// TwinCAT 3 PLC project TcoIoBeckhoffTests
// Title: TcoIoBeckhoffTests
// Company: Vortex.Library
// ProjectVersion: 1.19.1.1780
// ProgramVersion: 3.1.4024.12
// libraries:
//   Tc2_Standard, * (Beckhoff Automation GmbH)
//   Tc2_System, * (Beckhoff Automation GmbH)
//   Tc3_Module, * (Beckhoff Automation GmbH)
//   TcoCore, 1.19.1.1780 (Vortex.Library)
//   TcoIoBeckhoff, 1.19.1.1780 (Vortex.Library)
// project tree:
//   / PlcTask.TcTTO
//   POUs/ MAIN.TcPOU, tcc.TcPOU
//   DUTs/IO/PdoEntries/ Status_3D84275F.TcDUT (not stored), Ctrl_1EFB4D3B.TcDUT, Ctrl_71604E86.TcDUT, Status_B0753356.TcDUT, Status_F2CE6D91.TcDUT
//   DUTs/IO/PDOs/ COM_TxPDO_Map_Inputs_Channel_3801C95E.TcDUT, COM_RxPDO_Map_Outputs_Channel_EADA2E0D.TcDUT, WcState_9091E0EB.TcDUT, InfoData_32EB74EA.TcDUT (not stored), Channel_830843C1.TcDUT, InfoData_6F19DB2B.TcDUT, Channel_42CA91F7.TcDUT, AO_Outputs_Channel_BA7EBB7C.TcDUT, COM_Inputs_3801C95E.TcDUT, COM_Outputs_DEF408EC.TcDUT, PM_Inputs_Channel_2F868086.TcDUT, PM_Status_data_2A9514CB.TcDUT, PM_Outputs_Channel_E5FBDE30.TcDUT, AI_Standard_Channel_A8DF64E3.TcDUT, AI_Standard_4A394481.TcDUT, AI_Standard_Channel_4A394481.TcDUT
//   DUTs/IO/Boxes/ EL6002_81703A53.TcDUT, EL1809_32157CFD.TcDUT (not stored), EL2809_2B6483BD.TcDUT, EL4004_D2A7C9B7.TcDUT, EL6001_B592E1CA.TcDUT, EK1100_1FC0878B.TcDUT (not stored), EK1110_1FC0878B.TcDUT (not stored), EL3403_200C4240.TcDUT, EK1122_1FC0878B.TcDUT (not stored), EL3174_DCC78662.TcDUT (not stored), EL3011_353F32DF.TcDUT (not stored), EL2008_E2806B95.TcDUT, EL3024_C4269E32.TcDUT (not stored)
//   DUTs/IO/Devices/ SyncUnitTasks_1988CF1B.TcDUT, SyncUnits_13973095.TcDUT
//   DUTs/IO/Topology/ Term_1_EK1200_342ABB04.TcDUT (not stored), Device_1_EtherCAT_4442729B.TcDUT, Term_9_EK1100_B6B701E6.TcDUT, Term_17_EK1100_B932616E.TcDUT (not stored), Term_16_EK1122_E3300954.TcDUT (not stored), Term_14_EK1100_ED6DF06D.TcDUT (not stored), Device_4_EtherCAT_7DA382B8.TcDUT
//   GVLs/ GVL_iXlinker.TcGVL
// (motion and I/O tree: see PLC project tcoiobeckhoff)
// real-time tasks:
//   TASK PlcTask: cycle T#10ms, priority 20, ADS port 350
//   TASK PlcTask1: cycle T#10ms, priority 21, ADS port 351
//   TASK PlcTask2: cycle T#10ms, priority 22, ADS port 352
// variable links:
//   TcoIoBeckhoffTests/TcoIoBeckhoffTests Instance <-> Device 1 (EtherCAT)
//     PlcTask Inputs/GVL_iXlinker.Device_1_EtherCAT.InfoData.AmsNetId <-> InfoData/AmsNetId
//     PlcTask Inputs/GVL_iXlinker.Device_1_EtherCAT.InfoData.CfgSlaveCount <-> InfoData/CfgSlaveCount
//     PlcTask Inputs/GVL_iXlinker.Device_1_EtherCAT.InfoData.ChangeCount <-> InfoData/ChangeCount
//     PlcTask Inputs/GVL_iXlinker.Device_1_EtherCAT.InfoData.DevId <-> InfoData/DevId
//     PlcTask Inputs/GVL_iXlinker.Device_1_EtherCAT.Inputs.DevState <-> Inputs/DevState
//     PlcTask Inputs/GVL_iXlinker.Device_1_EtherCAT.Inputs.Frm0InputToggle <-> Inputs/Frm0InputToggle
//     PlcTask Inputs/GVL_iXlinker.Device_1_EtherCAT.Inputs.Frm0State <-> Inputs/Frm0State
//     PlcTask Inputs/GVL_iXlinker.Device_1_EtherCAT.Inputs.Frm0WcState <-> Inputs/Frm0WcState
//     PlcTask Inputs/GVL_iXlinker.Device_1_EtherCAT.Inputs.SlaveCount <-> Inputs/SlaveCount
//     PlcTask Inputs/GVL_iXlinker.Device_1_EtherCAT.SyncUnits._default.PlcTask1.InfoData.ObjectId <-> SyncUnits/<default>/PlcTask1/InfoData/ObjectId
//     PlcTask Inputs/GVL_iXlinker.Device_1_EtherCAT.SyncUnits._default.PlcTask1.InfoData.SlaveCount <-> SyncUnits/<default>/PlcTask1/InfoData/SlaveCount
//     PlcTask Inputs/GVL_iXlinker.Device_1_EtherCAT.SyncUnits._default.PlcTask1.InfoData.State <-> SyncUnits/<default>/PlcTask1/InfoData/State
//     PlcTask Inputs/GVL_iXlinker.Device_1_EtherCAT.SyncUnits._default.PlcTask1.WcState.WcState <-> SyncUnits/<default>/PlcTask1/WcState/WcState
//     PlcTask Outputs/GVL_iXlinker.Device_1_EtherCAT.Outputs.DevCtrl <-> Outputs/DevCtrl
//     PlcTask Outputs/GVL_iXlinker.Device_1_EtherCAT.Outputs.Frm0Ctrl <-> Outputs/Frm0Ctrl
//     PlcTask Outputs/GVL_iXlinker.Device_1_EtherCAT.Outputs.Frm0WcCtrl <-> Outputs/Frm0WcCtrl
//   TcoIoBeckhoffTests/TcoIoBeckhoffTests Instance <-> Device 1 (EtherCAT)/Term 1 (EK1200)/Term 2 (EL6002)
//     PlcTask Inputs/GVL_iXlinker.Device_1_EtherCAT.Term_1_EK1200.Term_2_EL6002.COM_TxPDO_Map_Inputs_Channel_1.Data_In[0] <-> COM TxPDO-Map Inputs Channel 1/Data In 0
//     PlcTask Inputs/GVL_iXlinker.Device_1_EtherCAT.Term_1_EK1200.Term_2_EL6002.COM_TxPDO_Map_Inputs_Channel_1.Data_In[10] <-> COM TxPDO-Map Inputs Channel 1/Data In 10
//     PlcTask Inputs/GVL_iXlinker.Device_1_EtherCAT.Term_1_EK1200.Term_2_EL6002.COM_TxPDO_Map_Inputs_Channel_1.Data_In[11] <-> COM TxPDO-Map Inputs Channel 1/Data In 11
//     PlcTask Inputs/GVL_iXlinker.Device_1_EtherCAT.Term_1_EK1200.Term_2_EL6002.COM_TxPDO_Map_Inputs_Channel_1.Data_In[12] <-> COM TxPDO-Map Inputs Channel 1/Data In 12
//     PlcTask Inputs/GVL_iXlinker.Device_1_EtherCAT.Term_1_EK1200.Term_2_EL6002.COM_TxPDO_Map_Inputs_Channel_1.Data_In[13] <-> COM TxPDO-Map Inputs Channel 1/Data In 13
//     PlcTask Inputs/GVL_iXlinker.Device_1_EtherCAT.Term_1_EK1200.Term_2_EL6002.COM_TxPDO_Map_Inputs_Channel_1.Data_In[14] <-> COM TxPDO-Map Inputs Channel 1/Data In 14
//     PlcTask Inputs/GVL_iXlinker.Device_1_EtherCAT.Term_1_EK1200.Term_2_EL6002.COM_TxPDO_Map_Inputs_Channel_1.Data_In[15] <-> COM TxPDO-Map Inputs Channel 1/Data In 15
//     PlcTask Inputs/GVL_iXlinker.Device_1_EtherCAT.Term_1_EK1200.Term_2_EL6002.COM_TxPDO_Map_Inputs_Channel_1.Data_In[16] <-> COM TxPDO-Map Inputs Channel 1/Data In 16
//     PlcTask Inputs/GVL_iXlinker.Device_1_EtherCAT.Term_1_EK1200.Term_2_EL6002.COM_TxPDO_Map_Inputs_Channel_1.Data_In[17] <-> COM TxPDO-Map Inputs Channel 1/Data In 17
//     PlcTask Inputs/GVL_iXlinker.Device_1_EtherCAT.Term_1_EK1200.Term_2_EL6002.COM_TxPDO_Map_Inputs_Channel_1.Data_In[18] <-> COM TxPDO-Map Inputs Channel 1/Data In 18
//     PlcTask Inputs/GVL_iXlinker.Device_1_EtherCAT.Term_1_EK1200.Term_2_EL6002.COM_TxPDO_Map_Inputs_Channel_1.Data_In[19] <-> COM TxPDO-Map Inputs Channel 1/Data In 19
//     PlcTask Inputs/GVL_iXlinker.Device_1_EtherCAT.Term_1_EK1200.Term_2_EL6002.COM_TxPDO_Map_Inputs_Channel_1.Data_In[1] <-> COM TxPDO-Map Inputs Channel 1/Data In 1
//     PlcTask Inputs/GVL_iXlinker.Device_1_EtherCAT.Term_1_EK1200.Term_2_EL6002.COM_TxPDO_Map_Inputs_Channel_1.Data_In[20] <-> COM TxPDO-Map Inputs Channel 1/Data In 20
//     PlcTask Inputs/GVL_iXlinker.Device_1_EtherCAT.Term_1_EK1200.Term_2_EL6002.COM_TxPDO_Map_Inputs_Channel_1.Data_In[21] <-> COM TxPDO-Map Inputs Channel 1/Data In 21
//     PlcTask Inputs/GVL_iXlinker.Device_1_EtherCAT.Term_1_EK1200.Term_2_EL6002.COM_TxPDO_Map_Inputs_Channel_1.Data_In[2] <-> COM TxPDO-Map Inputs Channel 1/Data In 2
//     PlcTask Inputs/GVL_iXlinker.Device_1_EtherCAT.Term_1_EK1200.Term_2_EL6002.COM_TxPDO_Map_Inputs_Channel_1.Data_In[3] <-> COM TxPDO-Map Inputs Channel 1/Data In 3
//     PlcTask Inputs/GVL_iXlinker.Device_1_EtherCAT.Term_1_EK1200.Term_2_EL6002.COM_TxPDO_Map_Inputs_Channel_1.Data_In[4] <-> COM TxPDO-Map Inputs Channel 1/Data In 4
//     PlcTask Inputs/GVL_iXlinker.Device_1_EtherCAT.Term_1_EK1200.Term_2_EL6002.COM_TxPDO_Map_Inputs_Channel_1.Data_In[5] <-> COM TxPDO-Map Inputs Channel 1/Data In 5
//     PlcTask Inputs/GVL_iXlinker.Device_1_EtherCAT.Term_1_EK1200.Term_2_EL6002.COM_TxPDO_Map_Inputs_Channel_1.Data_In[6] <-> COM TxPDO-Map Inputs Channel 1/Data In 6
//     PlcTask Inputs/GVL_iXlinker.Device_1_EtherCAT.Term_1_EK1200.Term_2_EL6002.COM_TxPDO_Map_Inputs_Channel_1.Data_In[7] <-> COM TxPDO-Map Inputs Channel 1/Data In 7
//     PlcTask Inputs/GVL_iXlinker.Device_1_EtherCAT.Term_1_EK1200.Term_2_EL6002.COM_TxPDO_Map_Inputs_Channel_1.Data_In[8] <-> COM TxPDO-Map Inputs Channel 1/Data In 8
//     PlcTask Inputs/GVL_iXlinker.Device_1_EtherCAT.Term_1_EK1200.Term_2_EL6002.COM_TxPDO_Map_Inputs_Channel_1.Data_In[9] <-> COM TxPDO-Map Inputs Channel 1/Data In 9
//     PlcTask Inputs/GVL_iXlinker.Device_1_EtherCAT.Term_1_EK1200.Term_2_EL6002.COM_TxPDO_Map_Inputs_Channel_2.Data_In[0] <-> COM TxPDO-Map Inputs Channel 2/Data In 0
//     PlcTask Inputs/GVL_iXlinker.Device_1_EtherCAT.Term_1_EK1200.Term_2_EL6002.COM_TxPDO_Map_Inputs_Channel_2.Data_In[10] <-> COM TxPDO-Map Inputs Channel 2/Data In 10
//     PlcTask Inputs/GVL_iXlinker.Device_1_EtherCAT.Term_1_EK1200.Term_2_EL6002.COM_TxPDO_Map_Inputs_Channel_2.Data_In[11] <-> COM TxPDO-Map Inputs Channel 2/Data In 11
//     PlcTask Inputs/GVL_iXlinker.Device_1_EtherCAT.Term_1_EK1200.Term_2_EL6002.COM_TxPDO_Map_Inputs_Channel_2.Data_In[12] <-> COM TxPDO-Map Inputs Channel 2/Data In 12
//     PlcTask Inputs/GVL_iXlinker.Device_1_EtherCAT.Term_1_EK1200.Term_2_EL6002.COM_TxPDO_Map_Inputs_Channel_2.Data_In[13] <-> COM TxPDO-Map Inputs Channel 2/Data In 13
//     PlcTask Inputs/GVL_iXlinker.Device_1_EtherCAT.Term_1_EK1200.Term_2_EL6002.COM_TxPDO_Map_Inputs_Channel_2.Data_In[14] <-> COM TxPDO-Map Inputs Channel 2/Data In 14
//     PlcTask Inputs/GVL_iXlinker.Device_1_EtherCAT.Term_1_EK1200.Term_2_EL6002.COM_TxPDO_Map_Inputs_Channel_2.Data_In[15] <-> COM TxPDO-Map Inputs Channel 2/Data In 15
//     PlcTask Inputs/GVL_iXlinker.Device_1_EtherCAT.Term_1_EK1200.Term_2_EL6002.COM_TxPDO_Map_Inputs_Channel_2.Data_In[16] <-> COM TxPDO-Map Inputs Channel 2/Data In 16
//     PlcTask Inputs/GVL_iXlinker.Device_1_EtherCAT.Term_1_EK1200.Term_2_EL6002.COM_TxPDO_Map_Inputs_Channel_2.Data_In[17] <-> COM TxPDO-Map Inputs Channel 2/Data In 17
//     PlcTask Inputs/GVL_iXlinker.Device_1_EtherCAT.Term_1_EK1200.Term_2_EL6002.COM_TxPDO_Map_Inputs_Channel_2.Data_In[18] <-> COM TxPDO-Map Inputs Channel 2/Data In 18
//     PlcTask Inputs/GVL_iXlinker.Device_1_EtherCAT.Term_1_EK1200.Term_2_EL6002.COM_TxPDO_Map_Inputs_Channel_2.Data_In[19] <-> COM TxPDO-Map Inputs Channel 2/Data In 19
//     PlcTask Inputs/GVL_iXlinker.Device_1_EtherCAT.Term_1_EK1200.Term_2_EL6002.COM_TxPDO_Map_Inputs_Channel_2.Data_In[1] <-> COM TxPDO-Map Inputs Channel 2/Data In 1
//     PlcTask Inputs/GVL_iXlinker.Device_1_EtherCAT.Term_1_EK1200.Term_2_EL6002.COM_TxPDO_Map_Inputs_Channel_2.Data_In[20] <-> COM TxPDO-Map Inputs Channel 2/Data In 20
//     PlcTask Inputs/GVL_iXlinker.Device_1_EtherCAT.Term_1_EK1200.Term_2_EL6002.COM_TxPDO_Map_Inputs_Channel_2.Data_In[21] <-> COM TxPDO-Map Inputs Channel 2/Data In 21
//     PlcTask Inputs/GVL_iXlinker.Device_1_EtherCAT.Term_1_EK1200.Term_2_EL6002.COM_TxPDO_Map_Inputs_Channel_2.Data_In[2] <-> COM TxPDO-Map Inputs Channel 2/Data In 2
//     PlcTask Inputs/GVL_iXlinker.Device_1_EtherCAT.Term_1_EK1200.Term_2_EL6002.COM_TxPDO_Map_Inputs_Channel_2.Data_In[3] <-> COM TxPDO-Map Inputs Channel 2/Data In 3
//     PlcTask Inputs/GVL_iXlinker.Device_1_EtherCAT.Term_1_EK1200.Term_2_EL6002.COM_TxPDO_Map_Inputs_Channel_2.Data_In[4] <-> COM TxPDO-Map Inputs Channel 2/Data In 4
//     PlcTask Inputs/GVL_iXlinker.Device_1_EtherCAT.Term_1_EK1200.Term_2_EL6002.COM_TxPDO_Map_Inputs_Channel_2.Data_In[5] <-> COM TxPDO-Map Inputs Channel 2/Data In 5
//     PlcTask Inputs/GVL_iXlinker.Device_1_EtherCAT.Term_1_EK1200.Term_2_EL6002.COM_TxPDO_Map_Inputs_Channel_2.Data_In[6] <-> COM TxPDO-Map Inputs Channel 2/Data In 6
//     PlcTask Inputs/GVL_iXlinker.Device_1_EtherCAT.Term_1_EK1200.Term_2_EL6002.COM_TxPDO_Map_Inputs_Channel_2.Data_In[7] <-> COM TxPDO-Map Inputs Channel 2/Data In 7
//     PlcTask Inputs/GVL_iXlinker.Device_1_EtherCAT.Term_1_EK1200.Term_2_EL6002.COM_TxPDO_Map_Inputs_Channel_2.Data_In[8] <-> COM TxPDO-Map Inputs Channel 2/Data In 8
//     PlcTask Inputs/GVL_iXlinker.Device_1_EtherCAT.Term_1_EK1200.Term_2_EL6002.COM_TxPDO_Map_Inputs_Channel_2.Data_In[9] <-> COM TxPDO-Map Inputs Channel 2/Data In 9
//     PlcTask Inputs/GVL_iXlinker.Device_1_EtherCAT.Term_1_EK1200.Term_2_EL6002.COM_TxPDO_Map_Inputs_Channel_1.Status/Buffer_full <-> COM TxPDO-Map Inputs Channel 1/Status/Buffer full
//     PlcTask Inputs/GVL_iXlinker.Device_1_EtherCAT.Term_1_EK1200.Term_2_EL6002.COM_TxPDO_Map_Inputs_Channel_2.Status/Buffer_full <-> COM TxPDO-Map Inputs Channel 2/Status/Buffer full
//     PlcTask Inputs/GVL_iXlinker.Device_1_EtherCAT.Term_1_EK1200.Term_2_EL6002.COM_TxPDO_Map_Inputs_Channel_1.Status/Framing_error <-> COM TxPDO-Map Inputs Channel 1/Status/Framing error
//     PlcTask Inputs/GVL_iXlinker.Device_1_EtherCAT.Term_1_EK1200.Term_2_EL6002.COM_TxPDO_Map_Inputs_Channel_2.Status/Framing_error <-> COM TxPDO-Map Inputs Channel 2/Status/Framing error
//     PlcTask Inputs/GVL_iXlinker.Device_1_EtherCAT.Term_1_EK1200.Term_2_EL6002.COM_TxPDO_Map_Inputs_Channel_1.Status/Init_accepted <-> COM TxPDO-Map Inputs Channel 1/Status/Init accepted
//     PlcTask Inputs/GVL_iXlinker.Device_1_EtherCAT.Term_1_EK1200.Term_2_EL6002.COM_TxPDO_Map_Inputs_Channel_2.Status/Init_accepted <-> COM TxPDO-Map Inputs Channel 2/Status/Init accepted
//     PlcTask Inputs/GVL_iXlinker.Device_1_EtherCAT.Term_1_EK1200.Term_2_EL6002.COM_TxPDO_Map_Inputs_Channel_1.Status/Input_length <-> COM TxPDO-Map Inputs Channel 1/Status/Input length
//     PlcTask Inputs/GVL_iXlinker.Device_1_EtherCAT.Term_1_EK1200.Term_2_EL6002.COM_TxPDO_Map_Inputs_Channel_2.Status/Input_length <-> COM TxPDO-Map Inputs Channel 2/Status/Input length
//     PlcTask Inputs/GVL_iXlinker.Device_1_EtherCAT.Term_1_EK1200.Term_2_EL6002.COM_TxPDO_Map_Inputs_Channel_1.Status/Overrun_error <-> COM TxPDO-Map Inputs Channel 1/Status/Overrun error
//     PlcTask Inputs/GVL_iXlinker.Device_1_EtherCAT.Term_1_EK1200.Term_2_EL6002.COM_TxPDO_Map_Inputs_Channel_2.Status/Overrun_error <-> COM TxPDO-Map Inputs Channel 2/Status/Overrun error
//     PlcTask Inputs/GVL_iXlinker.Device_1_EtherCAT.Term_1_EK1200.Term_2_EL6002.COM_TxPDO_Map_Inputs_Channel_1.Status/Parity_error <-> COM TxPDO-Map Inputs Channel 1/Status/Parity error
//     PlcTask Inputs/GVL_iXlinker.Device_1_EtherCAT.Term_1_EK1200.Term_2_EL6002.COM_TxPDO_Map_Inputs_Channel_2.Status/Parity_error <-> COM TxPDO-Map Inputs Channel 2/Status/Parity error
//     PlcTask Inputs/GVL_iXlinker.Device_1_EtherCAT.Term_1_EK1200.Term_2_EL6002.COM_TxPDO_Map_Inputs_Channel_1.Status/Receive_request <-> COM TxPDO-Map Inputs Channel 1/Status/Receive request
//     PlcTask Inputs/GVL_iXlinker.Device_1_EtherCAT.Term_1_EK1200.Term_2_EL6002.COM_TxPDO_Map_Inputs_Channel_2.Status/Receive_request <-> COM TxPDO-Map Inputs Channel 2/Status/Receive request
//     PlcTask Inputs/GVL_iXlinker.Device_1_EtherCAT.Term_1_EK1200.Term_2_EL6002.COM_TxPDO_Map_Inputs_Channel_1.Status/Transmit_accepted <-> COM TxPDO-Map Inputs Channel 1/Status/Transmit accepted
//     PlcTask Inputs/GVL_iXlinker.Device_1_EtherCAT.Term_1_EK1200.Term_2_EL6002.COM_TxPDO_Map_Inputs_Channel_2.Status/Transmit_accepted <-> COM TxPDO-Map Inputs Channel 2/Status/Transmit accepted
//     PlcTask Inputs/GVL_iXlinker.Device_1_EtherCAT.Term_1_EK1200.Term_2_EL6002.InfoData.State <-> InfoData/State
//     PlcTask Inputs/GVL_iXlinker.Device_1_EtherCAT.Term_1_EK1200.Term_2_EL6002.WcState.InputToggle <-> WcState/InputToggle
//     PlcTask Inputs/GVL_iXlinker.Device_1_EtherCAT.Term_1_EK1200.Term_2_EL6002.WcState.WcState <-> WcState/WcState
//     PlcTask Outputs/GVL_iXlinker.Device_1_EtherCAT.Term_1_EK1200.Term_2_EL6002.COM_RxPDO_Map_Outputs_Channel_1.Ctrl/Init_request <-> COM RxPDO-Map Outputs Channel 1/Ctrl/Init request
//     PlcTask Outputs/GVL_iXlinker.Device_1_EtherCAT.Term_1_EK1200.Term_2_EL6002.COM_RxPDO_Map_Outputs_Channel_2.Ctrl/Init_request <-> COM RxPDO-Map Outputs Channel 2/Ctrl/Init request
//     PlcTask Outputs/GVL_iXlinker.Device_1_EtherCAT.Term_1_EK1200.Term_2_EL6002.COM_RxPDO_Map_Outputs_Channel_1.Ctrl/Output_length <-> COM RxPDO-Map Outputs Channel 1/Ctrl/Output length
//     PlcTask Outputs/GVL_iXlinker.Device_1_EtherCAT.Term_1_EK1200.Term_2_EL6002.COM_RxPDO_Map_Outputs_Channel_2.Ctrl/Output_length <-> COM RxPDO-Map Outputs Channel 2/Ctrl/Output length
//     PlcTask Outputs/GVL_iXlinker.Device_1_EtherCAT.Term_1_EK1200.Term_2_EL6002.COM_RxPDO_Map_Outputs_Channel_1.Ctrl/Receive_accepted <-> COM RxPDO-Map Outputs Channel 1/Ctrl/Receive accepted
//     PlcTask Outputs/GVL_iXlinker.Device_1_EtherCAT.Term_1_EK1200.Term_2_EL6002.COM_RxPDO_Map_Outputs_Channel_2.Ctrl/Receive_accepted <-> COM RxPDO-Map Outputs Channel 2/Ctrl/Receive accepted
//     PlcTask Outputs/GVL_iXlinker.Device_1_EtherCAT.Term_1_EK1200.Term_2_EL6002.COM_RxPDO_Map_Outputs_Channel_1.Ctrl/Send_continuous <-> COM RxPDO-Map Outputs Channel 1/Ctrl/Send continuous
//     PlcTask Outputs/GVL_iXlinker.Device_1_EtherCAT.Term_1_EK1200.Term_2_EL6002.COM_RxPDO_Map_Outputs_Channel_2.Ctrl/Send_continuous <-> COM RxPDO-Map Outputs Channel 2/Ctrl/Send continuous
//     PlcTask Outputs/GVL_iXlinker.Device_1_EtherCAT.Term_1_EK1200.Term_2_EL6002.COM_RxPDO_Map_Outputs_Channel_1.Ctrl/Transmit_request <-> COM RxPDO-Map Outputs Channel 1/Ctrl/Transmit request
//     PlcTask Outputs/GVL_iXlinker.Device_1_EtherCAT.Term_1_EK1200.Term_2_EL6002.COM_RxPDO_Map_Outputs_Channel_2.Ctrl/Transmit_request <-> COM RxPDO-Map Outputs Channel 2/Ctrl/Transmit request
//     PlcTask Outputs/GVL_iXlinker.Device_1_EtherCAT.Term_1_EK1200.Term_2_EL6002.COM_RxPDO_Map_Outputs_Channel_1.Data_Out[0] <-> COM RxPDO-Map Outputs Channel 1/Data Out 0
//     PlcTask Outputs/GVL_iXlinker.Device_1_EtherCAT.Term_1_EK1200.Term_2_EL6002.COM_RxPDO_Map_Outputs_Channel_1.Data_Out[10] <-> COM RxPDO-Map Outputs Channel 1/Data Out 10
//     PlcTask Outputs/GVL_iXlinker.Device_1_EtherCAT.Term_1_EK1200.Term_2_EL6002.COM_RxPDO_Map_Outputs_Channel_1.Data_Out[11] <-> COM RxPDO-Map Outputs Channel 1/Data Out 11
//     PlcTask Outputs/GVL_iXlinker.Device_1_EtherCAT.Term_1_EK1200.Term_2_EL6002.COM_RxPDO_Map_Outputs_Channel_1.Data_Out[12] <-> COM RxPDO-Map Outputs Channel 1/Data Out 12
//     PlcTask Outputs/GVL_iXlinker.Device_1_EtherCAT.Term_1_EK1200.Term_2_EL6002.COM_RxPDO_Map_Outputs_Channel_1.Data_Out[13] <-> COM RxPDO-Map Outputs Channel 1/Data Out 13
//     PlcTask Outputs/GVL_iXlinker.Device_1_EtherCAT.Term_1_EK1200.Term_2_EL6002.COM_RxPDO_Map_Outputs_Channel_1.Data_Out[14] <-> COM RxPDO-Map Outputs Channel 1/Data Out 14
//     PlcTask Outputs/GVL_iXlinker.Device_1_EtherCAT.Term_1_EK1200.Term_2_EL6002.COM_RxPDO_Map_Outputs_Channel_1.Data_Out[15] <-> COM RxPDO-Map Outputs Channel 1/Data Out 15
//     PlcTask Outputs/GVL_iXlinker.Device_1_EtherCAT.Term_1_EK1200.Term_2_EL6002.COM_RxPDO_Map_Outputs_Channel_1.Data_Out[16] <-> COM RxPDO-Map Outputs Channel 1/Data Out 16
//     PlcTask Outputs/GVL_iXlinker.Device_1_EtherCAT.Term_1_EK1200.Term_2_EL6002.COM_RxPDO_Map_Outputs_Channel_1.Data_Out[17] <-> COM RxPDO-Map Outputs Channel 1/Data Out 17
//     PlcTask Outputs/GVL_iXlinker.Device_1_EtherCAT.Term_1_EK1200.Term_2_EL6002.COM_RxPDO_Map_Outputs_Channel_1.Data_Out[18] <-> COM RxPDO-Map Outputs Channel 1/Data Out 18
//     PlcTask Outputs/GVL_iXlinker.Device_1_EtherCAT.Term_1_EK1200.Term_2_EL6002.COM_RxPDO_Map_Outputs_Channel_1.Data_Out[19] <-> COM RxPDO-Map Outputs Channel 1/Data Out 19
//     PlcTask Outputs/GVL_iXlinker.Device_1_EtherCAT.Term_1_EK1200.Term_2_EL6002.COM_RxPDO_Map_Outputs_Channel_1.Data_Out[1] <-> COM RxPDO-Map Outputs Channel 1/Data Out 1
//     PlcTask Outputs/GVL_iXlinker.Device_1_EtherCAT.Term_1_EK1200.Term_2_EL6002.COM_RxPDO_Map_Outputs_Channel_1.Data_Out[20] <-> COM RxPDO-Map Outputs Channel 1/Data Out 20
//     PlcTask Outputs/GVL_iXlinker.Device_1_EtherCAT.Term_1_EK1200.Term_2_EL6002.COM_RxPDO_Map_Outputs_Channel_1.Data_Out[21] <-> COM RxPDO-Map Outputs Channel 1/Data Out 21
//     PlcTask Outputs/GVL_iXlinker.Device_1_EtherCAT.Term_1_EK1200.Term_2_EL6002.COM_RxPDO_Map_Outputs_Channel_1.Data_Out[2] <-> COM RxPDO-Map Outputs Channel 1/Data Out 2
//     PlcTask Outputs/GVL_iXlinker.Device_1_EtherCAT.Term_1_EK1200.Term_2_EL6002.COM_RxPDO_Map_Outputs_Channel_1.Data_Out[3] <-> COM RxPDO-Map Outputs Channel 1/Data Out 3
//     PlcTask Outputs/GVL_iXlinker.Device_1_EtherCAT.Term_1_EK1200.Term_2_EL6002.COM_RxPDO_Map_Outputs_Channel_1.Data_Out[4] <-> COM RxPDO-Map Outputs Channel 1/Data Out 4
//     PlcTask Outputs/GVL_iXlinker.Device_1_EtherCAT.Term_1_EK1200.Term_2_EL6002.COM_RxPDO_Map_Outputs_Channel_1.Data_Out[5] <-> COM RxPDO-Map Outputs Channel 1/Data Out 5
//     PlcTask Outputs/GVL_iXlinker.Device_1_EtherCAT.Term_1_EK1200.Term_2_EL6002.COM_RxPDO_Map_Outputs_Channel_1.Data_Out[6] <-> COM RxPDO-Map Outputs Channel 1/Data Out 6
//     PlcTask Outputs/GVL_iXlinker.Device_1_EtherCAT.Term_1_EK1200.Term_2_EL6002.COM_RxPDO_Map_Outputs_Channel_1.Data_Out[7] <-> COM RxPDO-Map Outputs Channel 1/Data Out 7
//     PlcTask Outputs/GVL_iXlinker.Device_1_EtherCAT.Term_1_EK1200.Term_2_EL6002.COM_RxPDO_Map_Outputs_Channel_1.Data_Out[8] <-> COM RxPDO-Map Outputs Channel 1/Data Out 8
//     PlcTask Outputs/GVL_iXlinker.Device_1_EtherCAT.Term_1_EK1200.Term_2_EL6002.COM_RxPDO_Map_Outputs_Channel_1.Data_Out[9] <-> COM RxPDO-Map Outputs Channel 1/Data Out 9
//     PlcTask Outputs/GVL_iXlinker.Device_1_EtherCAT.Term_1_EK1200.Term_2_EL6002.COM_RxPDO_Map_Outputs_Channel_2.Data_Out[0] <-> COM RxPDO-Map Outputs Channel 2/Data Out 0
//     PlcTask Outputs/GVL_iXlinker.Device_1_EtherCAT.Term_1_EK1200.Term_2_EL6002.COM_RxPDO_Map_Outputs_Channel_2.Data_Out[10] <-> COM RxPDO-Map Outputs Channel 2/Data Out 10
//     PlcTask Outputs/GVL_iXlinker.Device_1_EtherCAT.Term_1_EK1200.Term_2_EL6002.COM_RxPDO_Map_Outputs_Channel_2.Data_Out[11] <-> COM RxPDO-Map Outputs Channel 2/Data Out 11
//     PlcTask Outputs/GVL_iXlinker.Device_1_EtherCAT.Term_1_EK1200.Term_2_EL6002.COM_RxPDO_Map_Outputs_Channel_2.Data_Out[12] <-> COM RxPDO-Map Outputs Channel 2/Data Out 12
//     PlcTask Outputs/GVL_iXlinker.Device_1_EtherCAT.Term_1_EK1200.Term_2_EL6002.COM_RxPDO_Map_Outputs_Channel_2.Data_Out[13] <-> COM RxPDO-Map Outputs Channel 2/Data Out 13
//     PlcTask Outputs/GVL_iXlinker.Device_1_EtherCAT.Term_1_EK1200.Term_2_EL6002.COM_RxPDO_Map_Outputs_Channel_2.Data_Out[14] <-> COM RxPDO-Map Outputs Channel 2/Data Out 14
//     PlcTask Outputs/GVL_iXlinker.Device_1_EtherCAT.Term_1_EK1200.Term_2_EL6002.COM_RxPDO_Map_Outputs_Channel_2.Data_Out[15] <-> COM RxPDO-Map Outputs Channel 2/Data Out 15
//     PlcTask Outputs/GVL_iXlinker.Device_1_EtherCAT.Term_1_EK1200.Term_2_EL6002.COM_RxPDO_Map_Outputs_Channel_2.Data_Out[16] <-> COM RxPDO-Map Outputs Channel 2/Data Out 16
//     PlcTask Outputs/GVL_iXlinker.Device_1_EtherCAT.Term_1_EK1200.Term_2_EL6002.COM_RxPDO_Map_Outputs_Channel_2.Data_Out[17] <-> COM RxPDO-Map Outputs Channel 2/Data Out 17
//     PlcTask Outputs/GVL_iXlinker.Device_1_EtherCAT.Term_1_EK1200.Term_2_EL6002.COM_RxPDO_Map_Outputs_Channel_2.Data_Out[18] <-> COM RxPDO-Map Outputs Channel 2/Data Out 18
//     PlcTask Outputs/GVL_iXlinker.Device_1_EtherCAT.Term_1_EK1200.Term_2_EL6002.COM_RxPDO_Map_Outputs_Channel_2.Data_Out[19] <-> COM RxPDO-Map Outputs Channel 2/Data Out 19
//     PlcTask Outputs/GVL_iXlinker.Device_1_EtherCAT.Term_1_EK1200.Term_2_EL6002.COM_RxPDO_Map_Outputs_Channel_2.Data_Out[1] <-> COM RxPDO-Map Outputs Channel 2/Data Out 1
//     PlcTask Outputs/GVL_iXlinker.Device_1_EtherCAT.Term_1_EK1200.Term_2_EL6002.COM_RxPDO_Map_Outputs_Channel_2.Data_Out[20] <-> COM RxPDO-Map Outputs Channel 2/Data Out 20
//     PlcTask Outputs/GVL_iXlinker.Device_1_EtherCAT.Term_1_EK1200.Term_2_EL6002.COM_RxPDO_Map_Outputs_Channel_2.Data_Out[21] <-> COM RxPDO-Map Outputs Channel 2/Data Out 21
//     PlcTask Outputs/GVL_iXlinker.Device_1_EtherCAT.Term_1_EK1200.Term_2_EL6002.COM_RxPDO_Map_Outputs_Channel_2.Data_Out[2] <-> COM RxPDO-Map Outputs Channel 2/Data Out 2
//     PlcTask Outputs/GVL_iXlinker.Device_1_EtherCAT.Term_1_EK1200.Term_2_EL6002.COM_RxPDO_Map_Outputs_Channel_2.Data_Out[3] <-> COM RxPDO-Map Outputs Channel 2/Data Out 3
//     PlcTask Outputs/GVL_iXlinker.Device_1_EtherCAT.Term_1_EK1200.Term_2_EL6002.COM_RxPDO_Map_Outputs_Channel_2.Data_Out[4] <-> COM RxPDO-Map Outputs Channel 2/Data Out 4
//     PlcTask Outputs/GVL_iXlinker.Device_1_EtherCAT.Term_1_EK1200.Term_2_EL6002.COM_RxPDO_Map_Outputs_Channel_2.Data_Out[5] <-> COM RxPDO-Map Outputs Channel 2/Data Out 5
//     PlcTask Outputs/GVL_iXlinker.Device_1_EtherCAT.Term_1_EK1200.Term_2_EL6002.COM_RxPDO_Map_Outputs_Channel_2.Data_Out[6] <-> COM RxPDO-Map Outputs Channel 2/Data Out 6
//     PlcTask Outputs/GVL_iXlinker.Device_1_EtherCAT.Term_1_EK1200.Term_2_EL6002.COM_RxPDO_Map_Outputs_Channel_2.Data_Out[7] <-> COM RxPDO-Map Outputs Channel 2/Data Out 7
//     PlcTask Outputs/GVL_iXlinker.Device_1_EtherCAT.Term_1_EK1200.Term_2_EL6002.COM_RxPDO_Map_Outputs_Channel_2.Data_Out[8] <-> COM RxPDO-Map Outputs Channel 2/Data Out 8
//     PlcTask Outputs/GVL_iXlinker.Device_1_EtherCAT.Term_1_EK1200.Term_2_EL6002.COM_RxPDO_Map_Outputs_Channel_2.Data_Out[9] <-> COM RxPDO-Map Outputs Channel 2/Data Out 9
//   TcoIoBeckhoffTests/TcoIoBeckhoffTests Instance <-> Device 1 (EtherCAT)/Term 1 (EK1200)/Term 3 (EL1809)
//     PlcTask Inputs/GVL_iXlinker.Device_1_EtherCAT.Term_1_EK1200.Term_3_EL1809.Channel_{1..16}.Input <-> Channel {1..16}/Input  (16 links)
//     PlcTask Inputs/GVL_iXlinker.Device_1_EtherCAT.Term_1_EK1200.Term_3_EL1809.InfoData.State <-> InfoData/State
//     PlcTask Inputs/GVL_iXlinker.Device_1_EtherCAT.Term_1_EK1200.Term_3_EL1809.WcState.InputToggle <-> WcState/InputToggle
//     PlcTask Inputs/GVL_iXlinker.Device_1_EtherCAT.Term_1_EK1200.Term_3_EL1809.WcState.WcState <-> WcState/WcState
//   TcoIoBeckhoffTests/TcoIoBeckhoffTests Instance <-> Device 1 (EtherCAT)/Term 1 (EK1200)/Term 4 (EL2809)
//     PlcTask Inputs/GVL_iXlinker.Device_1_EtherCAT.Term_1_EK1200.Term_4_EL2809.InfoData.State <-> InfoData/State
//     PlcTask Inputs/GVL_iXlinker.Device_1_EtherCAT.Term_1_EK1200.Term_4_EL2809.WcState.WcState <-> WcState/WcState
//     PlcTask Outputs/GVL_iXlinker.Device_1_EtherCAT.Term_1_EK1200.Term_4_EL2809.Channel_{1..16}.Output <-> Channel {1..16}/Output  (16 links)
//   TcoIoBeckhoffTests/TcoIoBeckhoffTests Instance <-> Device 1 (EtherCAT)/Term 1 (EK1200)/Term 5 (EL4004)
//     PlcTask Inputs/GVL_iXlinker.Device_1_EtherCAT.Term_1_EK1200.Term_5_EL4004.InfoData.State <-> InfoData/State
//     PlcTask Inputs/GVL_iXlinker.Device_1_EtherCAT.Term_1_EK1200.Term_5_EL4004.WcState.WcState <-> WcState/WcState
//     PlcTask Outputs/GVL_iXlinker.Device_1_EtherCAT.Term_1_EK1200.Term_5_EL4004.AO_Outputs_Channel_{1..4}.Analog_output <-> AO Outputs Channel {1..4}/Analog output  (4 links)
//   TcoIoBeckhoffTests/TcoIoBeckhoffTests Instance <-> Device 1 (EtherCAT)/Term 1 (EK1200)/Term 6 (EL2809)
//     PlcTask Inputs/GVL_iXlinker.Device_1_EtherCAT.Term_1_EK1200.Term_6_EL2809.InfoData.State <-> InfoData/State
//     PlcTask Inputs/GVL_iXlinker.Device_1_EtherCAT.Term_1_EK1200.Term_6_EL2809.WcState.WcState <-> WcState/WcState
//     PlcTask Outputs/GVL_iXlinker.Device_1_EtherCAT.Term_1_EK1200.Term_6_EL2809.Channel_{1..16}.Output <-> Channel {1..16}/Output  (16 links)
//   TcoIoBeckhoffTests/TcoIoBeckhoffTests Instance <-> Device 1 (EtherCAT)/Term 1 (EK1200)/Term 7 (EL6001)
//     PlcTask Inputs/GVL_iXlinker.Device_1_EtherCAT.Term_1_EK1200.Term_7_EL6001.COM_Inputs.Data_In[{0..21}] <-> COM Inputs/Data In {0..21}  (22 links)
//     PlcTask Inputs/GVL_iXlinker.Device_1_EtherCAT.Term_1_EK1200.Term_7_EL6001.COM_Inputs.Status/Buffer_full <-> COM Inputs/Status/Buffer full
//     PlcTask Inputs/GVL_iXlinker.Device_1_EtherCAT.Term_1_EK1200.Term_7_EL6001.COM_Inputs.Status/Framing_error <-> COM Inputs/Status/Framing error
//     PlcTask Inputs/GVL_iXlinker.Device_1_EtherCAT.Term_1_EK1200.Term_7_EL6001.COM_Inputs.Status/Init_accepted <-> COM Inputs/Status/Init accepted
//     PlcTask Inputs/GVL_iXlinker.Device_1_EtherCAT.Term_1_EK1200.Term_7_EL6001.COM_Inputs.Status/Input_length <-> COM Inputs/Status/Input length
//     PlcTask Inputs/GVL_iXlinker.Device_1_EtherCAT.Term_1_EK1200.Term_7_EL6001.COM_Inputs.Status/Overrun_error <-> COM Inputs/Status/Overrun error
//     PlcTask Inputs/GVL_iXlinker.Device_1_EtherCAT.Term_1_EK1200.Term_7_EL6001.COM_Inputs.Status/Parity_error <-> COM Inputs/Status/Parity error
//     PlcTask Inputs/GVL_iXlinker.Device_1_EtherCAT.Term_1_EK1200.Term_7_EL6001.COM_Inputs.Status/Receive_request <-> COM Inputs/Status/Receive request
//     PlcTask Inputs/GVL_iXlinker.Device_1_EtherCAT.Term_1_EK1200.Term_7_EL6001.COM_Inputs.Status/Transmit_accepted <-> COM Inputs/Status/Transmit accepted
//     PlcTask Inputs/GVL_iXlinker.Device_1_EtherCAT.Term_1_EK1200.Term_7_EL6001.InfoData.State <-> InfoData/State
//     PlcTask Inputs/GVL_iXlinker.Device_1_EtherCAT.Term_1_EK1200.Term_7_EL6001.WcState.InputToggle <-> WcState/InputToggle
//     PlcTask Inputs/GVL_iXlinker.Device_1_EtherCAT.Term_1_EK1200.Term_7_EL6001.WcState.WcState <-> WcState/WcState
//     PlcTask Outputs/GVL_iXlinker.Device_1_EtherCAT.Term_1_EK1200.Term_7_EL6001.COM_Outputs.Ctrl/Init_request <-> COM Outputs/Ctrl/Init request
//     PlcTask Outputs/GVL_iXlinker.Device_1_EtherCAT.Term_1_EK1200.Term_7_EL6001.COM_Outputs.Ctrl/Output_length <-> COM Outputs/Ctrl/Output length
//     PlcTask Outputs/GVL_iXlinker.Device_1_EtherCAT.Term_1_EK1200.Term_7_EL6001.COM_Outputs.Ctrl/Receive_accepted <-> COM Outputs/Ctrl/Receive accepted
//     PlcTask Outputs/GVL_iXlinker.Device_1_EtherCAT.Term_1_EK1200.Term_7_EL6001.COM_Outputs.Ctrl/Send_continues <-> COM Outputs/Ctrl/Send continues
//     PlcTask Outputs/GVL_iXlinker.Device_1_EtherCAT.Term_1_EK1200.Term_7_EL6001.COM_Outputs.Ctrl/Transmit_request <-> COM Outputs/Ctrl/Transmit request
//     PlcTask Outputs/GVL_iXlinker.Device_1_EtherCAT.Term_1_EK1200.Term_7_EL6001.COM_Outputs.Data_Out[{0..21}] <-> COM Outputs/Data Out {0..21}  (22 links)
//   TcoIoBeckhoffTests/TcoIoBeckhoffTests Instance <-> Device 4 (EtherCAT)
//     PlcTask Inputs/GVL_iXlinker.Device_4_EtherCAT.InfoData.AmsNetId <-> InfoData/AmsNetId
//     PlcTask Inputs/GVL_iXlinker.Device_4_EtherCAT.InfoData.CfgSlaveCount <-> InfoData/CfgSlaveCount
//     PlcTask Inputs/GVL_iXlinker.Device_4_EtherCAT.InfoData.ChangeCount <-> InfoData/ChangeCount
//     PlcTask Inputs/GVL_iXlinker.Device_4_EtherCAT.InfoData.DevId <-> InfoData/DevId
//     PlcTask Inputs/GVL_iXlinker.Device_4_EtherCAT.Inputs.DevState <-> Inputs/DevState
//     PlcTask Inputs/GVL_iXlinker.Device_4_EtherCAT.Inputs.Frm0InputToggle <-> Inputs/Frm0InputToggle
//     PlcTask Inputs/GVL_iXlinker.Device_4_EtherCAT.Inputs.Frm0State <-> Inputs/Frm0State
//     PlcTask Inputs/GVL_iXlinker.Device_4_EtherCAT.Inputs.Frm0WcState <-> Inputs/Frm0WcState
//     PlcTask Inputs/GVL_iXlinker.Device_4_EtherCAT.Inputs.SlaveCount <-> Inputs/SlaveCount
//     PlcTask Inputs/GVL_iXlinker.Device_4_EtherCAT.SyncUnits._default.PlcTask1.InfoData.ObjectId <-> SyncUnits/<default>/PlcTask1/InfoData/ObjectId
//     PlcTask Inputs/GVL_iXlinker.Device_4_EtherCAT.SyncUnits._default.PlcTask1.InfoData.SlaveCount <-> SyncUnits/<default>/PlcTask1/InfoData/SlaveCount
//     PlcTask Inputs/GVL_iXlinker.Device_4_EtherCAT.SyncUnits._default.PlcTask1.InfoData.State <-> SyncUnits/<default>/PlcTask1/InfoData/State
//     PlcTask Inputs/GVL_iXlinker.Device_4_EtherCAT.SyncUnits._default.PlcTask1.WcState.WcState <-> SyncUnits/<default>/PlcTask1/WcState/WcState
//     PlcTask Outputs/GVL_iXlinker.Device_4_EtherCAT.Outputs.DevCtrl <-> Outputs/DevCtrl
//     PlcTask Outputs/GVL_iXlinker.Device_4_EtherCAT.Outputs.Frm0Ctrl <-> Outputs/Frm0Ctrl
//     PlcTask Outputs/GVL_iXlinker.Device_4_EtherCAT.Outputs.Frm0WcCtrl <-> Outputs/Frm0WcCtrl
//   TcoIoBeckhoffTests/TcoIoBeckhoffTests Instance <-> Device 4 (EtherCAT)/Term 14 (EK1100)
//     PlcTask Inputs/GVL_iXlinker.Device_4_EtherCAT.Term_14_EK1100.InfoData.State <-> InfoData/State
//   TcoIoBeckhoffTests/TcoIoBeckhoffTests Instance <-> Device 4 (EtherCAT)/Term 14 (EK1100)/Term 15 (EL3403)
//     PlcTask Inputs/GVL_iXlinker.Device_4_EtherCAT.Term_14_EK1100.Term_15_EL3403.InfoData.AdsAddr <-> InfoData/AdsAddr
//     PlcTask Inputs/GVL_iXlinker.Device_4_EtherCAT.Term_14_EK1100.Term_15_EL3403.InfoData.State <-> InfoData/State
//     PlcTask Inputs/GVL_iXlinker.Device_4_EtherCAT.Term_14_EK1100.Term_15_EL3403.PM_Inputs_Channel_1.Active_power <-> PM Inputs Channel 1/Active power
//     PlcTask Inputs/GVL_iXlinker.Device_4_EtherCAT.Term_14_EK1100.Term_15_EL3403.PM_Inputs_Channel_2.Active_power <-> PM Inputs Channel 2/Active power
//     PlcTask Inputs/GVL_iXlinker.Device_4_EtherCAT.Term_14_EK1100.Term_15_EL3403.PM_Inputs_Channel_3.Active_power <-> PM Inputs Channel 3/Active power
//     PlcTask Inputs/GVL_iXlinker.Device_4_EtherCAT.Term_14_EK1100.Term_15_EL3403.PM_Inputs_Channel_1.Current <-> PM Inputs Channel 1/Current
//     PlcTask Inputs/GVL_iXlinker.Device_4_EtherCAT.Term_14_EK1100.Term_15_EL3403.PM_Inputs_Channel_2.Current <-> PM Inputs Channel 2/Current
//     PlcTask Inputs/GVL_iXlinker.Device_4_EtherCAT.Term_14_EK1100.Term_15_EL3403.PM_Inputs_Channel_3.Current <-> PM Inputs Channel 3/Current
//     PlcTask Inputs/GVL_iXlinker.Device_4_EtherCAT.Term_14_EK1100.Term_15_EL3403.PM_Inputs_Channel_1.Index <-> PM Inputs Channel 1/Index
//     PlcTask Inputs/GVL_iXlinker.Device_4_EtherCAT.Term_14_EK1100.Term_15_EL3403.PM_Inputs_Channel_2.Index <-> PM Inputs Channel 2/Index
//     PlcTask Inputs/GVL_iXlinker.Device_4_EtherCAT.Term_14_EK1100.Term_15_EL3403.PM_Inputs_Channel_3.Index <-> PM Inputs Channel 3/Index
//     PlcTask Inputs/GVL_iXlinker.Device_4_EtherCAT.Term_14_EK1100.Term_15_EL3403.PM_Inputs_Channel_1.TxPDO_Toggle <-> PM Inputs Channel 1/TxPDO Toggle
//     PlcTask Inputs/GVL_iXlinker.Device_4_EtherCAT.Term_14_EK1100.Term_15_EL3403.PM_Inputs_Channel_2.TxPDO_Toggle <-> PM Inputs Channel 2/TxPDO Toggle
//     PlcTask Inputs/GVL_iXlinker.Device_4_EtherCAT.Term_14_EK1100.Term_15_EL3403.PM_Inputs_Channel_3.TxPDO_Toggle <-> PM Inputs Channel 3/TxPDO Toggle
//     PlcTask Inputs/GVL_iXlinker.Device_4_EtherCAT.Term_14_EK1100.Term_15_EL3403.PM_Inputs_Channel_1.Variant_value <-> PM Inputs Channel 1/Variant value
//     PlcTask Inputs/GVL_iXlinker.Device_4_EtherCAT.Term_14_EK1100.Term_15_EL3403.PM_Inputs_Channel_2.Variant_value <-> PM Inputs Channel 2/Variant value
//     PlcTask Inputs/GVL_iXlinker.Device_4_EtherCAT.Term_14_EK1100.Term_15_EL3403.PM_Inputs_Channel_3.Variant_value <-> PM Inputs Channel 3/Variant value
//     PlcTask Inputs/GVL_iXlinker.Device_4_EtherCAT.Term_14_EK1100.Term_15_EL3403.PM_Inputs_Channel_1.Voltage <-> PM Inputs Channel 1/Voltage
//     PlcTask Inputs/GVL_iXlinker.Device_4_EtherCAT.Term_14_EK1100.Term_15_EL3403.PM_Inputs_Channel_2.Voltage <-> PM Inputs Channel 2/Voltage
//     PlcTask Inputs/GVL_iXlinker.Device_4_EtherCAT.Term_14_EK1100.Term_15_EL3403.PM_Inputs_Channel_3.Voltage <-> PM Inputs Channel 3/Voltage
//     PlcTask Inputs/GVL_iXlinker.Device_4_EtherCAT.Term_14_EK1100.Term_15_EL3403.PM_Status_data.Missing_zero_crossing_A <-> PM Status data/Missing zero crossing A
//     PlcTask Inputs/GVL_iXlinker.Device_4_EtherCAT.Term_14_EK1100.Term_15_EL3403.PM_Status_data.Missing_zero_crossing_B <-> PM Status data/Missing zero crossing B
//     PlcTask Inputs/GVL_iXlinker.Device_4_EtherCAT.Term_14_EK1100.Term_15_EL3403.PM_Status_data.Missing_zero_crossing_C <-> PM Status data/Missing zero crossing C
//     PlcTask Inputs/GVL_iXlinker.Device_4_EtherCAT.Term_14_EK1100.Term_15_EL3403.PM_Status_data.Phase_sequence_error <-> PM Status data/Phase sequence error
//     PlcTask Inputs/GVL_iXlinker.Device_4_EtherCAT.Term_14_EK1100.Term_15_EL3403.WcState.InputToggle <-> WcState/InputToggle
//     PlcTask Inputs/GVL_iXlinker.Device_4_EtherCAT.Term_14_EK1100.Term_15_EL3403.WcState.WcState <-> WcState/WcState
//     PlcTask Outputs/GVL_iXlinker.Device_4_EtherCAT.Term_14_EK1100.Term_15_EL3403.PM_Outputs_Channel_1.Index <-> PM Outputs Channel 1/Index
//     PlcTask Outputs/GVL_iXlinker.Device_4_EtherCAT.Term_14_EK1100.Term_15_EL3403.PM_Outputs_Channel_2.Index <-> PM Outputs Channel 2/Index
//     PlcTask Outputs/GVL_iXlinker.Device_4_EtherCAT.Term_14_EK1100.Term_15_EL3403.PM_Outputs_Channel_3.Index <-> PM Outputs Channel 3/Index
//   TcoIoBeckhoffTests/TcoIoBeckhoffTests Instance <-> Device 4 (EtherCAT)/Term 14 (EK1100)/Term 16 (EK1122)
//     PlcTask Inputs/GVL_iXlinker.Device_4_EtherCAT.Term_14_EK1100.Term_16_EK1122.InfoData.State <-> InfoData/State
//   TcoIoBeckhoffTests/TcoIoBeckhoffTests Instance <-> Device 4 (EtherCAT)/Term 14 (EK1100)/Term 16 (EK1122)/Term 17 (EK1100)
//     PlcTask Inputs/GVL_iXlinker.Device_4_EtherCAT.Term_14_EK1100.Term_16_EK1122.Term_17_EK1100.InfoData.State <-> InfoData/State
//   TcoIoBeckhoffTests/TcoIoBeckhoffTests Instance <-> Device 4 (EtherCAT)/Term 14 (EK1100)/Term 16 (EK1122)/Term 17 (EK1100)/Term 18 (EL3174-0002)
//     PlcTask Inputs/GVL_iXlinker.Device_4_EtherCAT.Term_14_EK1100.Term_16_EK1122.Term_17_EK1100.Term_18_EL3174_0002.AI_Standard_Channel_1.Status/Error <-> AI Standard Channel 1/Status/Error
//     PlcTask Inputs/GVL_iXlinker.Device_4_EtherCAT.Term_14_EK1100.Term_16_EK1122.Term_17_EK1100.Term_18_EL3174_0002.AI_Standard_Channel_2.Status/Error <-> AI Standard Channel 2/Status/Error
//     PlcTask Inputs/GVL_iXlinker.Device_4_EtherCAT.Term_14_EK1100.Term_16_EK1122.Term_17_EK1100.Term_18_EL3174_0002.AI_Standard_Channel_3.Status/Error <-> AI Standard Channel 3/Status/Error
//     PlcTask Inputs/GVL_iXlinker.Device_4_EtherCAT.Term_14_EK1100.Term_16_EK1122.Term_17_EK1100.Term_18_EL3174_0002.AI_Standard_Channel_4.Status/Error <-> AI Standard Channel 4/Status/Error
//     PlcTask Inputs/GVL_iXlinker.Device_4_EtherCAT.Term_14_EK1100.Term_16_EK1122.Term_17_EK1100.Term_18_EL3174_0002.AI_Standard_Channel_1.Status/Limit_1 <-> AI Standard Channel 1/Status/Limit 1
//     PlcTask Inputs/GVL_iXlinker.Device_4_EtherCAT.Term_14_EK1100.Term_16_EK1122.Term_17_EK1100.Term_18_EL3174_0002.AI_Standard_Channel_1.Status/Limit_2 <-> AI Standard Channel 1/Status/Limit 2
//     PlcTask Inputs/GVL_iXlinker.Device_4_EtherCAT.Term_14_EK1100.Term_16_EK1122.Term_17_EK1100.Term_18_EL3174_0002.AI_Standard_Channel_2.Status/Limit_1 <-> AI Standard Channel 2/Status/Limit 1
//     PlcTask Inputs/GVL_iXlinker.Device_4_EtherCAT.Term_14_EK1100.Term_16_EK1122.Term_17_EK1100.Term_18_EL3174_0002.AI_Standard_Channel_2.Status/Limit_2 <-> AI Standard Channel 2/Status/Limit 2
//     PlcTask Inputs/GVL_iXlinker.Device_4_EtherCAT.Term_14_EK1100.Term_16_EK1122.Term_17_EK1100.Term_18_EL3174_0002.AI_Standard_Channel_3.Status/Limit_1 <-> AI Standard Channel 3/Status/Limit 1
//     PlcTask Inputs/GVL_iXlinker.Device_4_EtherCAT.Term_14_EK1100.Term_16_EK1122.Term_17_EK1100.Term_18_EL3174_0002.AI_Standard_Channel_3.Status/Limit_2 <-> AI Standard Channel 3/Status/Limit 2
//     PlcTask Inputs/GVL_iXlinker.Device_4_EtherCAT.Term_14_EK1100.Term_16_EK1122.Term_17_EK1100.Term_18_EL3174_0002.AI_Standard_Channel_4.Status/Limit_1 <-> AI Standard Channel 4/Status/Limit 1
//     PlcTask Inputs/GVL_iXlinker.Device_4_EtherCAT.Term_14_EK1100.Term_16_EK1122.Term_17_EK1100.Term_18_EL3174_0002.AI_Standard_Channel_4.Status/Limit_2 <-> AI Standard Channel 4/Status/Limit 2
//     PlcTask Inputs/GVL_iXlinker.Device_4_EtherCAT.Term_14_EK1100.Term_16_EK1122.Term_17_EK1100.Term_18_EL3174_0002.AI_Standard_Channel_1.Status/Overrange <-> AI Standard Channel 1/Status/Overrange
//     PlcTask Inputs/GVL_iXlinker.Device_4_EtherCAT.Term_14_EK1100.Term_16_EK1122.Term_17_EK1100.Term_18_EL3174_0002.AI_Standard_Channel_2.Status/Overrange <-> AI Standard Channel 2/Status/Overrange
//     PlcTask Inputs/GVL_iXlinker.Device_4_EtherCAT.Term_14_EK1100.Term_16_EK1122.Term_17_EK1100.Term_18_EL3174_0002.AI_Standard_Channel_3.Status/Overrange <-> AI Standard Channel 3/Status/Overrange
//     PlcTask Inputs/GVL_iXlinker.Device_4_EtherCAT.Term_14_EK1100.Term_16_EK1122.Term_17_EK1100.Term_18_EL3174_0002.AI_Standard_Channel_4.Status/Overrange <-> AI Standard Channel 4/Status/Overrange
//     PlcTask Inputs/GVL_iXlinker.Device_4_EtherCAT.Term_14_EK1100.Term_16_EK1122.Term_17_EK1100.Term_18_EL3174_0002.AI_Standard_Channel_1.Status/Sync_error <-> AI Standard Channel 1/Status/Sync error
//     PlcTask Inputs/GVL_iXlinker.Device_4_EtherCAT.Term_14_EK1100.Term_16_EK1122.Term_17_EK1100.Term_18_EL3174_0002.AI_Standard_Channel_2.Status/Sync_error <-> AI Standard Channel 2/Status/Sync error
//     PlcTask Inputs/GVL_iXlinker.Device_4_EtherCAT.Term_14_EK1100.Term_16_EK1122.Term_17_EK1100.Term_18_EL3174_0002.AI_Standard_Channel_3.Status/Sync_error <-> AI Standard Channel 3/Status/Sync error
//     PlcTask Inputs/GVL_iXlinker.Device_4_EtherCAT.Term_14_EK1100.Term_16_EK1122.Term_17_EK1100.Term_18_EL3174_0002.AI_Standard_Channel_4.Status/Sync_error <-> AI Standard Channel 4/Status/Sync error
//     PlcTask Inputs/GVL_iXlinker.Device_4_EtherCAT.Term_14_EK1100.Term_16_EK1122.Term_17_EK1100.Term_18_EL3174_0002.AI_Standard_Channel_1.Status/TxPDO_State <-> AI Standard Channel 1/Status/TxPDO State
//     PlcTask Inputs/GVL_iXlinker.Device_4_EtherCAT.Term_14_EK1100.Term_16_EK1122.Term_17_EK1100.Term_18_EL3174_0002.AI_Standard_Channel_2.Status/TxPDO_State <-> AI Standard Channel 2/Status/TxPDO State
//     PlcTask Inputs/GVL_iXlinker.Device_4_EtherCAT.Term_14_EK1100.Term_16_EK1122.Term_17_EK1100.Term_18_EL3174_0002.AI_Standard_Channel_3.Status/TxPDO_State <-> AI Standard Channel 3/Status/TxPDO State
//     PlcTask Inputs/GVL_iXlinker.Device_4_EtherCAT.Term_14_EK1100.Term_16_EK1122.Term_17_EK1100.Term_18_EL3174_0002.AI_Standard_Channel_4.Status/TxPDO_State <-> AI Standard Channel 4/Status/TxPDO State
//     PlcTask Inputs/GVL_iXlinker.Device_4_EtherCAT.Term_14_EK1100.Term_16_EK1122.Term_17_EK1100.Term_18_EL3174_0002.AI_Standard_Channel_1.Status/TxPDO_Toggle <-> AI Standard Channel 1/Status/TxPDO Toggle
//     PlcTask Inputs/GVL_iXlinker.Device_4_EtherCAT.Term_14_EK1100.Term_16_EK1122.Term_17_EK1100.Term_18_EL3174_0002.AI_Standard_Channel_2.Status/TxPDO_Toggle <-> AI Standard Channel 2/Status/TxPDO Toggle
//     PlcTask Inputs/GVL_iXlinker.Device_4_EtherCAT.Term_14_EK1100.Term_16_EK1122.Term_17_EK1100.Term_18_EL3174_0002.AI_Standard_Channel_3.Status/TxPDO_Toggle <-> AI Standard Channel 3/Status/TxPDO Toggle
//     PlcTask Inputs/GVL_iXlinker.Device_4_EtherCAT.Term_14_EK1100.Term_16_EK1122.Term_17_EK1100.Term_18_EL3174_0002.AI_Standard_Channel_4.Status/TxPDO_Toggle <-> AI Standard Channel 4/Status/TxPDO Toggle
//     PlcTask Inputs/GVL_iXlinker.Device_4_EtherCAT.Term_14_EK1100.Term_16_EK1122.Term_17_EK1100.Term_18_EL3174_0002.AI_Standard_Channel_1.Status/Underrange <-> AI Standard Channel 1/Status/Underrange
//     PlcTask Inputs/GVL_iXlinker.Device_4_EtherCAT.Term_14_EK1100.Term_16_EK1122.Term_17_EK1100.Term_18_EL3174_0002.AI_Standard_Channel_2.Status/Underrange <-> AI Standard Channel 2/Status/Underrange
//     PlcTask Inputs/GVL_iXlinker.Device_4_EtherCAT.Term_14_EK1100.Term_16_EK1122.Term_17_EK1100.Term_18_EL3174_0002.AI_Standard_Channel_3.Status/Underrange <-> AI Standard Channel 3/Status/Underrange
//     PlcTask Inputs/GVL_iXlinker.Device_4_EtherCAT.Term_14_EK1100.Term_16_EK1122.Term_17_EK1100.Term_18_EL3174_0002.AI_Standard_Channel_4.Status/Underrange <-> AI Standard Channel 4/Status/Underrange
//     PlcTask Inputs/GVL_iXlinker.Device_4_EtherCAT.Term_14_EK1100.Term_16_EK1122.Term_17_EK1100.Term_18_EL3174_0002.AI_Standard_Channel_1.Value <-> AI Standard Channel 1/Value
//     PlcTask Inputs/GVL_iXlinker.Device_4_EtherCAT.Term_14_EK1100.Term_16_EK1122.Term_17_EK1100.Term_18_EL3174_0002.AI_Standard_Channel_2.Value <-> AI Standard Channel 2/Value
//     PlcTask Inputs/GVL_iXlinker.Device_4_EtherCAT.Term_14_EK1100.Term_16_EK1122.Term_17_EK1100.Term_18_EL3174_0002.AI_Standard_Channel_3.Value <-> AI Standard Channel 3/Value
//     PlcTask Inputs/GVL_iXlinker.Device_4_EtherCAT.Term_14_EK1100.Term_16_EK1122.Term_17_EK1100.Term_18_EL3174_0002.AI_Standard_Channel_4.Value <-> AI Standard Channel 4/Value
//     PlcTask Inputs/GVL_iXlinker.Device_4_EtherCAT.Term_14_EK1100.Term_16_EK1122.Term_17_EK1100.Term_18_EL3174_0002.InfoData.AdsAddr <-> InfoData/AdsAddr
//     PlcTask Inputs/GVL_iXlinker.Device_4_EtherCAT.Term_14_EK1100.Term_16_EK1122.Term_17_EK1100.Term_18_EL3174_0002.InfoData.State <-> InfoData/State
//     PlcTask Inputs/GVL_iXlinker.Device_4_EtherCAT.Term_14_EK1100.Term_16_EK1122.Term_17_EK1100.Term_18_EL3174_0002.WcState.InputToggle <-> WcState/InputToggle
//     PlcTask Inputs/GVL_iXlinker.Device_4_EtherCAT.Term_14_EK1100.Term_16_EK1122.Term_17_EK1100.Term_18_EL3174_0002.WcState.WcState <-> WcState/WcState
//   TcoIoBeckhoffTests/TcoIoBeckhoffTests Instance <-> Device 4 (EtherCAT)/Term 14 (EK1100)/Term 16 (EK1122)/Term 17 (EK1100)/Term 19 (EL6001)
//     PlcTask Inputs/GVL_iXlinker.Device_4_EtherCAT.Term_14_EK1100.Term_16_EK1122.Term_17_EK1100.Term_19_EL6001.COM_Inputs.Data_In[{0..21}] <-> COM Inputs/Data In {0..21}  (22 links)
//     PlcTask Inputs/GVL_iXlinker.Device_4_EtherCAT.Term_14_EK1100.Term_16_EK1122.Term_17_EK1100.Term_19_EL6001.COM_Inputs.Status/Buffer_full <-> COM Inputs/Status/Buffer full
//     PlcTask Inputs/GVL_iXlinker.Device_4_EtherCAT.Term_14_EK1100.Term_16_EK1122.Term_17_EK1100.Term_19_EL6001.COM_Inputs.Status/Framing_error <-> COM Inputs/Status/Framing error
//     PlcTask Inputs/GVL_iXlinker.Device_4_EtherCAT.Term_14_EK1100.Term_16_EK1122.Term_17_EK1100.Term_19_EL6001.COM_Inputs.Status/Init_accepted <-> COM Inputs/Status/Init accepted
//     PlcTask Inputs/GVL_iXlinker.Device_4_EtherCAT.Term_14_EK1100.Term_16_EK1122.Term_17_EK1100.Term_19_EL6001.COM_Inputs.Status/Input_length <-> COM Inputs/Status/Input length
//     PlcTask Inputs/GVL_iXlinker.Device_4_EtherCAT.Term_14_EK1100.Term_16_EK1122.Term_17_EK1100.Term_19_EL6001.COM_Inputs.Status/Overrun_error <-> COM Inputs/Status/Overrun error
//     PlcTask Inputs/GVL_iXlinker.Device_4_EtherCAT.Term_14_EK1100.Term_16_EK1122.Term_17_EK1100.Term_19_EL6001.COM_Inputs.Status/Parity_error <-> COM Inputs/Status/Parity error
//     PlcTask Inputs/GVL_iXlinker.Device_4_EtherCAT.Term_14_EK1100.Term_16_EK1122.Term_17_EK1100.Term_19_EL6001.COM_Inputs.Status/Receive_request <-> COM Inputs/Status/Receive request
//     PlcTask Inputs/GVL_iXlinker.Device_4_EtherCAT.Term_14_EK1100.Term_16_EK1122.Term_17_EK1100.Term_19_EL6001.COM_Inputs.Status/Transmit_accepted <-> COM Inputs/Status/Transmit accepted
//     PlcTask Inputs/GVL_iXlinker.Device_4_EtherCAT.Term_14_EK1100.Term_16_EK1122.Term_17_EK1100.Term_19_EL6001.InfoData.AdsAddr <-> InfoData/AdsAddr
//     PlcTask Inputs/GVL_iXlinker.Device_4_EtherCAT.Term_14_EK1100.Term_16_EK1122.Term_17_EK1100.Term_19_EL6001.InfoData.State <-> InfoData/State
//     PlcTask Inputs/GVL_iXlinker.Device_4_EtherCAT.Term_14_EK1100.Term_16_EK1122.Term_17_EK1100.Term_19_EL6001.WcState.InputToggle <-> WcState/InputToggle
//     PlcTask Inputs/GVL_iXlinker.Device_4_EtherCAT.Term_14_EK1100.Term_16_EK1122.Term_17_EK1100.Term_19_EL6001.WcState.WcState <-> WcState/WcState
//     PlcTask Outputs/GVL_iXlinker.Device_4_EtherCAT.Term_14_EK1100.Term_16_EK1122.Term_17_EK1100.Term_19_EL6001.COM_Outputs.Ctrl/Init_request <-> COM Outputs/Ctrl/Init request
//     PlcTask Outputs/GVL_iXlinker.Device_4_EtherCAT.Term_14_EK1100.Term_16_EK1122.Term_17_EK1100.Term_19_EL6001.COM_Outputs.Ctrl/Output_length <-> COM Outputs/Ctrl/Output length
//     PlcTask Outputs/GVL_iXlinker.Device_4_EtherCAT.Term_14_EK1100.Term_16_EK1122.Term_17_EK1100.Term_19_EL6001.COM_Outputs.Ctrl/Receive_accepted <-> COM Outputs/Ctrl/Receive accepted
//     PlcTask Outputs/GVL_iXlinker.Device_4_EtherCAT.Term_14_EK1100.Term_16_EK1122.Term_17_EK1100.Term_19_EL6001.COM_Outputs.Ctrl/Send_continues <-> COM Outputs/Ctrl/Send continues
//     PlcTask Outputs/GVL_iXlinker.Device_4_EtherCAT.Term_14_EK1100.Term_16_EK1122.Term_17_EK1100.Term_19_EL6001.COM_Outputs.Ctrl/Transmit_request <-> COM Outputs/Ctrl/Transmit request
//     PlcTask Outputs/GVL_iXlinker.Device_4_EtherCAT.Term_14_EK1100.Term_16_EK1122.Term_17_EK1100.Term_19_EL6001.COM_Outputs.Data_Out[{0..21}] <-> COM Outputs/Data Out {0..21}  (22 links)
//   TcoIoBeckhoffTests/TcoIoBeckhoffTests Instance <-> Device 4 (EtherCAT)/Term 14 (EK1100)/Term 16 (EK1122)/Term 17 (EK1100)/Term 20 (EL3011)
//     PlcTask Inputs/GVL_iXlinker.Device_4_EtherCAT.Term_14_EK1100.Term_16_EK1122.Term_17_EK1100.Term_20_EL3011.AI_Standard.Status/Error <-> AI Standard/Status/Error
//     PlcTask Inputs/GVL_iXlinker.Device_4_EtherCAT.Term_14_EK1100.Term_16_EK1122.Term_17_EK1100.Term_20_EL3011.AI_Standard.Status/Limit_1 <-> AI Standard/Status/Limit 1
//     PlcTask Inputs/GVL_iXlinker.Device_4_EtherCAT.Term_14_EK1100.Term_16_EK1122.Term_17_EK1100.Term_20_EL3011.AI_Standard.Status/Limit_2 <-> AI Standard/Status/Limit 2
//     PlcTask Inputs/GVL_iXlinker.Device_4_EtherCAT.Term_14_EK1100.Term_16_EK1122.Term_17_EK1100.Term_20_EL3011.AI_Standard.Status/Overrange <-> AI Standard/Status/Overrange
//     PlcTask Inputs/GVL_iXlinker.Device_4_EtherCAT.Term_14_EK1100.Term_16_EK1122.Term_17_EK1100.Term_20_EL3011.AI_Standard.Status/TxPDO_State <-> AI Standard/Status/TxPDO State
//     PlcTask Inputs/GVL_iXlinker.Device_4_EtherCAT.Term_14_EK1100.Term_16_EK1122.Term_17_EK1100.Term_20_EL3011.AI_Standard.Status/TxPDO_Toggle <-> AI Standard/Status/TxPDO Toggle
//     PlcTask Inputs/GVL_iXlinker.Device_4_EtherCAT.Term_14_EK1100.Term_16_EK1122.Term_17_EK1100.Term_20_EL3011.AI_Standard.Status/Underrange <-> AI Standard/Status/Underrange
//     PlcTask Inputs/GVL_iXlinker.Device_4_EtherCAT.Term_14_EK1100.Term_16_EK1122.Term_17_EK1100.Term_20_EL3011.AI_Standard.Value <-> AI Standard/Value
//     PlcTask Inputs/GVL_iXlinker.Device_4_EtherCAT.Term_14_EK1100.Term_16_EK1122.Term_17_EK1100.Term_20_EL3011.InfoData.AdsAddr <-> InfoData/AdsAddr
//     PlcTask Inputs/GVL_iXlinker.Device_4_EtherCAT.Term_14_EK1100.Term_16_EK1122.Term_17_EK1100.Term_20_EL3011.InfoData.State <-> InfoData/State
//     PlcTask Inputs/GVL_iXlinker.Device_4_EtherCAT.Term_14_EK1100.Term_16_EK1122.Term_17_EK1100.Term_20_EL3011.WcState.InputToggle <-> WcState/InputToggle
//     PlcTask Inputs/GVL_iXlinker.Device_4_EtherCAT.Term_14_EK1100.Term_16_EK1122.Term_17_EK1100.Term_20_EL3011.WcState.WcState <-> WcState/WcState
//   TcoIoBeckhoffTests/TcoIoBeckhoffTests Instance <-> Device 4 (EtherCAT)/Term 14 (EK1100)/Term 16 (EK1122)/Term 17 (EK1100)/Term 21 (EL2008)
//     PlcTask Inputs/GVL_iXlinker.Device_4_EtherCAT.Term_14_EK1100.Term_16_EK1122.Term_17_EK1100.Term_21_EL2008.InfoData.State <-> InfoData/State
//     PlcTask Inputs/GVL_iXlinker.Device_4_EtherCAT.Term_14_EK1100.Term_16_EK1122.Term_17_EK1100.Term_21_EL2008.WcState.WcState <-> WcState/WcState
//     PlcTask Outputs/GVL_iXlinker.Device_4_EtherCAT.Term_14_EK1100.Term_16_EK1122.Term_17_EK1100.Term_21_EL2008.Channel_{1..8}.Output <-> Channel {1..8}/Output  (8 links)
//   TcoIoBeckhoffTests/TcoIoBeckhoffTests Instance <-> Device 4 (EtherCAT)/Term 14 (EK1100)/Term 16 (EK1122)/Term 17 (EK1100)/Term 22 (EL2008)
//     PlcTask Inputs/GVL_iXlinker.Device_4_EtherCAT.Term_14_EK1100.Term_16_EK1122.Term_17_EK1100.Term_22_EL2008.InfoData.State <-> InfoData/State
//     PlcTask Inputs/GVL_iXlinker.Device_4_EtherCAT.Term_14_EK1100.Term_16_EK1122.Term_17_EK1100.Term_22_EL2008.WcState.WcState <-> WcState/WcState
//     PlcTask Outputs/GVL_iXlinker.Device_4_EtherCAT.Term_14_EK1100.Term_16_EK1122.Term_17_EK1100.Term_22_EL2008.Channel_{1..8}.Output <-> Channel {1..8}/Output  (8 links)
//   TcoIoBeckhoffTests/TcoIoBeckhoffTests Instance <-> Device 4 (EtherCAT)/Term 14 (EK1100)/Term 23 (EL3024)
//     PlcTask Inputs/GVL_iXlinker.Device_4_EtherCAT.Term_14_EK1100.Term_23_EL3024.AI_Standard_Channel_{1..4}.Status/Error <-> AI Standard Channel {1..4}/Status/Error  (4 links)
//     PlcTask Inputs/GVL_iXlinker.Device_4_EtherCAT.Term_14_EK1100.Term_23_EL3024.AI_Standard_Channel_1.Status/Limit_1 <-> AI Standard Channel 1/Status/Limit 1
//     PlcTask Inputs/GVL_iXlinker.Device_4_EtherCAT.Term_14_EK1100.Term_23_EL3024.AI_Standard_Channel_1.Status/Limit_2 <-> AI Standard Channel 1/Status/Limit 2
//     PlcTask Inputs/GVL_iXlinker.Device_4_EtherCAT.Term_14_EK1100.Term_23_EL3024.AI_Standard_Channel_2.Status/Limit_1 <-> AI Standard Channel 2/Status/Limit 1
//     PlcTask Inputs/GVL_iXlinker.Device_4_EtherCAT.Term_14_EK1100.Term_23_EL3024.AI_Standard_Channel_2.Status/Limit_2 <-> AI Standard Channel 2/Status/Limit 2
//     PlcTask Inputs/GVL_iXlinker.Device_4_EtherCAT.Term_14_EK1100.Term_23_EL3024.AI_Standard_Channel_3.Status/Limit_1 <-> AI Standard Channel 3/Status/Limit 1
//     PlcTask Inputs/GVL_iXlinker.Device_4_EtherCAT.Term_14_EK1100.Term_23_EL3024.AI_Standard_Channel_3.Status/Limit_2 <-> AI Standard Channel 3/Status/Limit 2
//     PlcTask Inputs/GVL_iXlinker.Device_4_EtherCAT.Term_14_EK1100.Term_23_EL3024.AI_Standard_Channel_4.Status/Limit_1 <-> AI Standard Channel 4/Status/Limit 1
//     PlcTask Inputs/GVL_iXlinker.Device_4_EtherCAT.Term_14_EK1100.Term_23_EL3024.AI_Standard_Channel_4.Status/Limit_2 <-> AI Standard Channel 4/Status/Limit 2
//     PlcTask Inputs/GVL_iXlinker.Device_4_EtherCAT.Term_14_EK1100.Term_23_EL3024.AI_Standard_Channel_{1..4}.Status/Overrange <-> AI Standard Channel {1..4}/Status/Overrange  (4 links)
//     PlcTask Inputs/GVL_iXlinker.Device_4_EtherCAT.Term_14_EK1100.Term_23_EL3024.AI_Standard_Channel_{1..4}.Status/TxPDO_State <-> AI Standard Channel {1..4}/Status/TxPDO State  (4 links)
//     PlcTask Inputs/GVL_iXlinker.Device_4_EtherCAT.Term_14_EK1100.Term_23_EL3024.AI_Standard_Channel_{1..4}.Status/TxPDO_Toggle <-> AI Standard Channel {1..4}/Status/TxPDO Toggle  (4 links)
//     PlcTask Inputs/GVL_iXlinker.Device_4_EtherCAT.Term_14_EK1100.Term_23_EL3024.AI_Standard_Channel_{1..4}.Status/Underrange <-> AI Standard Channel {1..4}/Status/Underrange  (4 links)
//     PlcTask Inputs/GVL_iXlinker.Device_4_EtherCAT.Term_14_EK1100.Term_23_EL3024.AI_Standard_Channel_{1..4}.Value <-> AI Standard Channel {1..4}/Value  (4 links)
//     PlcTask Inputs/GVL_iXlinker.Device_4_EtherCAT.Term_14_EK1100.Term_23_EL3024.InfoData.AdsAddr <-> InfoData/AdsAddr
//     PlcTask Inputs/GVL_iXlinker.Device_4_EtherCAT.Term_14_EK1100.Term_23_EL3024.InfoData.State <-> InfoData/State
//     PlcTask Inputs/GVL_iXlinker.Device_4_EtherCAT.Term_14_EK1100.Term_23_EL3024.WcState.InputToggle <-> WcState/InputToggle
//     PlcTask Inputs/GVL_iXlinker.Device_4_EtherCAT.Term_14_EK1100.Term_23_EL3024.WcState.WcState <-> WcState/WcState
//   TcoIoBeckhoffTests/TcoIoBeckhoffTests Instance <-> Device 4 (EtherCAT)/Term 9 (EK1100)
//     PlcTask Inputs/GVL_iXlinker.Device_4_EtherCAT.Term_9_EK1100.InfoData.State <-> InfoData/State
//   TcoIoBeckhoffTests/TcoIoBeckhoffTests Instance <-> Device 4 (EtherCAT)/Term 9 (EK1100)/Term 10 (EL6001)
//     PlcTask Inputs/GVL_iXlinker.Device_4_EtherCAT.Term_9_EK1100.Term_10_EL6001.COM_Inputs.Data_In[{0..21}] <-> COM Inputs/Data In {0..21}  (22 links)
//     PlcTask Inputs/GVL_iXlinker.Device_4_EtherCAT.Term_9_EK1100.Term_10_EL6001.COM_Inputs.Status/Buffer_full <-> COM Inputs/Status/Buffer full
//     PlcTask Inputs/GVL_iXlinker.Device_4_EtherCAT.Term_9_EK1100.Term_10_EL6001.COM_Inputs.Status/Framing_error <-> COM Inputs/Status/Framing error
//     PlcTask Inputs/GVL_iXlinker.Device_4_EtherCAT.Term_9_EK1100.Term_10_EL6001.COM_Inputs.Status/Init_accepted <-> COM Inputs/Status/Init accepted
//     PlcTask Inputs/GVL_iXlinker.Device_4_EtherCAT.Term_9_EK1100.Term_10_EL6001.COM_Inputs.Status/Input_length <-> COM Inputs/Status/Input length
//     PlcTask Inputs/GVL_iXlinker.Device_4_EtherCAT.Term_9_EK1100.Term_10_EL6001.COM_Inputs.Status/Overrun_error <-> COM Inputs/Status/Overrun error
//     PlcTask Inputs/GVL_iXlinker.Device_4_EtherCAT.Term_9_EK1100.Term_10_EL6001.COM_Inputs.Status/Parity_error <-> COM Inputs/Status/Parity error
//     PlcTask Inputs/GVL_iXlinker.Device_4_EtherCAT.Term_9_EK1100.Term_10_EL6001.COM_Inputs.Status/Receive_request <-> COM Inputs/Status/Receive request
//     PlcTask Inputs/GVL_iXlinker.Device_4_EtherCAT.Term_9_EK1100.Term_10_EL6001.COM_Inputs.Status/Transmit_accepted <-> COM Inputs/Status/Transmit accepted
//     PlcTask Inputs/GVL_iXlinker.Device_4_EtherCAT.Term_9_EK1100.Term_10_EL6001.InfoData.AdsAddr <-> InfoData/AdsAddr
//     PlcTask Inputs/GVL_iXlinker.Device_4_EtherCAT.Term_9_EK1100.Term_10_EL6001.InfoData.State <-> InfoData/State
//     PlcTask Inputs/GVL_iXlinker.Device_4_EtherCAT.Term_9_EK1100.Term_10_EL6001.WcState.InputToggle <-> WcState/InputToggle
//     PlcTask Inputs/GVL_iXlinker.Device_4_EtherCAT.Term_9_EK1100.Term_10_EL6001.WcState.WcState <-> WcState/WcState
//     PlcTask Outputs/GVL_iXlinker.Device_4_EtherCAT.Term_9_EK1100.Term_10_EL6001.COM_Outputs.Ctrl/Init_request <-> COM Outputs/Ctrl/Init request
//     PlcTask Outputs/GVL_iXlinker.Device_4_EtherCAT.Term_9_EK1100.Term_10_EL6001.COM_Outputs.Ctrl/Output_length <-> COM Outputs/Ctrl/Output length
//     PlcTask Outputs/GVL_iXlinker.Device_4_EtherCAT.Term_9_EK1100.Term_10_EL6001.COM_Outputs.Ctrl/Receive_accepted <-> COM Outputs/Ctrl/Receive accepted
//     PlcTask Outputs/GVL_iXlinker.Device_4_EtherCAT.Term_9_EK1100.Term_10_EL6001.COM_Outputs.Ctrl/Send_continues <-> COM Outputs/Ctrl/Send continues
//     PlcTask Outputs/GVL_iXlinker.Device_4_EtherCAT.Term_9_EK1100.Term_10_EL6001.COM_Outputs.Ctrl/Transmit_request <-> COM Outputs/Ctrl/Transmit request
//     PlcTask Outputs/GVL_iXlinker.Device_4_EtherCAT.Term_9_EK1100.Term_10_EL6001.COM_Outputs.Data_Out[{0..21}] <-> COM Outputs/Data Out {0..21}  (22 links)
//   TcoIoBeckhoffTests/TcoIoBeckhoffTests Instance <-> Device 4 (EtherCAT)/Term 9 (EK1100)/Term 11 (EL1809)
//     PlcTask Inputs/GVL_iXlinker.Device_4_EtherCAT.Term_9_EK1100.Term_11_EL1809.Channel_{1..16}.Input <-> Channel {1..16}/Input  (16 links)
//     PlcTask Inputs/GVL_iXlinker.Device_4_EtherCAT.Term_9_EK1100.Term_11_EL1809.InfoData.State <-> InfoData/State
//     PlcTask Inputs/GVL_iXlinker.Device_4_EtherCAT.Term_9_EK1100.Term_11_EL1809.WcState.InputToggle <-> WcState/InputToggle
//     PlcTask Inputs/GVL_iXlinker.Device_4_EtherCAT.Term_9_EK1100.Term_11_EL1809.WcState.WcState <-> WcState/WcState
//   TcoIoBeckhoffTests/TcoIoBeckhoffTests Instance <-> Device 4 (EtherCAT)/Term 9 (EK1100)/Term 12 (EL2809)
//     PlcTask Inputs/GVL_iXlinker.Device_4_EtherCAT.Term_9_EK1100.Term_12_EL2809.InfoData.State <-> InfoData/State
//     PlcTask Inputs/GVL_iXlinker.Device_4_EtherCAT.Term_9_EK1100.Term_12_EL2809.WcState.WcState <-> WcState/WcState
//     PlcTask Outputs/GVL_iXlinker.Device_4_EtherCAT.Term_9_EK1100.Term_12_EL2809.Channel_{1..16}.Output <-> Channel {1..16}/Output  (16 links)
//   TcoIoBeckhoffTests/TcoIoBeckhoffTests Instance <-> Device 4 (EtherCAT)/Term 9 (EK1100)/Term 13 (EK1110)
//     PlcTask Inputs/GVL_iXlinker.Device_4_EtherCAT.Term_9_EK1100.Term_13_EK1110.InfoData.State <-> InfoData/State

CONFIGURATION TcoIoBeckhoffTests
    RESOURCE PLC ON TwinCAT3
        TASK PlcTask(INTERVAL := T#10ms, PRIORITY := 21);
        PROGRAM MAIN WITH PlcTask : MAIN;
    END_RESOURCE
END_CONFIGURATION

// ---- DUTs/IO/PdoEntries/Ctrl_1EFB4D3B.TcDUT
{attribute 'GeneratedUsingTerminal: EL6002-0000-0019'}
{attribute addProperty BoxType "EL6002-0000-0019"}
{attribute addProperty Id "Transmit_requestBOOL1Receive_acceptedBOOL1Init_requestBOOL1Send_continuousBOOL1Output_lengthUSINT1"}
{attribute addProperty CRC "519785787"}
{attribute addProperty Size "5"}
TYPE Ctrl_1EFB4D3B :
STRUCT
	{attribute addProperty Name "Transmit_request"}
	Transmit_request : BOOL;
	{attribute addProperty Name "Receive_accepted"}
	Receive_accepted : BOOL;
	{attribute addProperty Name "Init_request"}
	Init_request : BOOL;
	{attribute addProperty Name "Send_continuous"}
	Send_continuous : BOOL;
	{attribute addProperty Name "Output_length"}
	Output_length : USINT;
END_STRUCT
END_TYPE

// ---- DUTs/IO/PdoEntries/Ctrl_71604E86.TcDUT
{attribute 'GeneratedUsingTerminal: EL6001-0000-0020'}
{attribute addProperty BoxType "EL6001-0000-0020"}
{attribute addProperty Id "Transmit_requestBOOL1Receive_acceptedBOOL1Init_requestBOOL1Send_continuesBOOL1Output_lengthUSINT1"}
{attribute addProperty CRC "1902136966"}
{attribute addProperty Size "5"}
TYPE Ctrl_71604E86 :
STRUCT
	{attribute addProperty Name "Transmit_request"}
	Transmit_request : BOOL;
	{attribute addProperty Name "Receive_accepted"}
	Receive_accepted : BOOL;
	{attribute addProperty Name "Init_request"}
	Init_request : BOOL;
	{attribute addProperty Name "Send_continues"}
	Send_continues : BOOL;
	{attribute addProperty Name "Output_length"}
	Output_length : USINT;
END_STRUCT
END_TYPE

// ---- DUTs/IO/PdoEntries/Status_B0753356.TcDUT
{attribute 'GeneratedUsingTerminal: EL3174-0002-0017'}
{attribute addProperty BoxType "EL3174-0002-0017"}
{attribute addProperty Id "UnderrangeBOOL1OverrangeBOOL1Limit_1BYTE1Limit_2BYTE1ErrorBOOL1Sync_errorBOOL1TxPDO_StateBOOL1TxPDO_ToggleBOOL1"}
{attribute addProperty CRC "2960470870"}
{attribute addProperty Size "8"}
TYPE Status_B0753356 :
STRUCT
	{attribute addProperty Name "Underrange"}
	Underrange : BOOL;
	{attribute addProperty Name "Overrange"}
	Overrange : BOOL;
	{attribute addProperty Name "Limit_1"}
	Limit_1 : BYTE;
	{attribute addProperty Name "Limit_2"}
	Limit_2 : BYTE;
	{attribute addProperty Name "Error"}
	Error : BOOL;
	{attribute addProperty Name "Sync_error"}
	Sync_error : BOOL;
	{attribute addProperty Name "TxPDO_State"}
	TxPDO_State : BOOL;
	{attribute addProperty Name "TxPDO_Toggle"}
	TxPDO_Toggle : BOOL;
END_STRUCT
END_TYPE

// ---- DUTs/IO/PdoEntries/Status_F2CE6D91.TcDUT
{attribute 'GeneratedUsingTerminal: EL3011-0000-0018'}
{attribute addProperty BoxType "EL3011-0000-0018"}
{attribute addProperty Id "UnderrangeBOOL1OverrangeBOOL1Limit_1BYTE1Limit_2BYTE1ErrorBOOL1TxPDO_StateBOOL1TxPDO_ToggleBOOL1"}
{attribute addProperty CRC "4073614737"}
{attribute addProperty Size "7"}
TYPE Status_F2CE6D91 :
STRUCT
	{attribute addProperty Name "Underrange"}
	Underrange : BOOL;
	{attribute addProperty Name "Overrange"}
	Overrange : BOOL;
	{attribute addProperty Name "Limit_1"}
	Limit_1 : BYTE;
	{attribute addProperty Name "Limit_2"}
	Limit_2 : BYTE;
	{attribute addProperty Name "Error"}
	Error : BOOL;
	{attribute addProperty Name "TxPDO_State"}
	TxPDO_State : BOOL;
	{attribute addProperty Name "TxPDO_Toggle"}
	TxPDO_Toggle : BOOL;
END_STRUCT
END_TYPE

// ---- DUTs/IO/PDOs/COM_TxPDO_Map_Inputs_Channel_3801C95E.TcDUT
{attribute 'GeneratedUsingTerminal: EL6002-0000-0019'}
{attribute addProperty BoxType "EL6002-0000-0019"}
{attribute addProperty Id "StatusAT %I*Status_3D84275F8Data_InAT %I*ARRAY[0..21] OF USINT22"}
{attribute addProperty CRC "1334739266"}
{attribute addProperty Size "30"}
TYPE COM_TxPDO_Map_Inputs_Channel_3801C95E :
STRUCT
	{attribute addProperty Name "Status"}
	Status AT %I* : Status_3D84275F;
	{attribute addProperty Name "Data_In"}
	Data_In AT %I* : ARRAY[0..21] OF USINT;
END_STRUCT
END_TYPE

// ---- DUTs/IO/PDOs/COM_RxPDO_Map_Outputs_Channel_EADA2E0D.TcDUT
{attribute 'GeneratedUsingTerminal: EL6002-0000-0019'}
{attribute addProperty BoxType "EL6002-0000-0019"}
{attribute addProperty Id "CtrlAT %Q*Ctrl_1EFB4D3B5Data_OutAT %Q*ARRAY[0..21] OF USINT22"}
{attribute addProperty CRC "3494673196"}
{attribute addProperty Size "27"}
TYPE COM_RxPDO_Map_Outputs_Channel_EADA2E0D :
STRUCT
	{attribute addProperty Name "Ctrl"}
	Ctrl AT %Q* : Ctrl_1EFB4D3B;
	{attribute addProperty Name "Data_Out"}
	Data_Out AT %Q* : ARRAY[0..21] OF USINT;
END_STRUCT
END_TYPE

// ---- DUTs/IO/PDOs/WcState_9091E0EB.TcDUT
{attribute 'GeneratedUsingTerminal: EL6002-0000-0019'}
{attribute addProperty BoxType "EL6002-0000-0019"}
{attribute addProperty Id "WcStateAT %I*BOOL1InputToggleAT %I*BOOL1"}
{attribute addProperty CRC "2425479403"}
{attribute addProperty Size "2"}
TYPE WcState_9091E0EB :
STRUCT
	{attribute addProperty Name "WcState"}
	WcState AT %I* : BOOL;
	{attribute addProperty Name "InputToggle"}
	InputToggle AT %I* : BOOL;
END_STRUCT
END_TYPE

// ---- DUTs/IO/PDOs/Channel_830843C1.TcDUT
{attribute 'GeneratedUsingTerminal: EL1809-0000-0018'}
{attribute addProperty BoxType "EL1809-0000-0018"}
{attribute addProperty Id "InputAT %I*BOOL1"}
{attribute addProperty CRC "2198356929"}
{attribute addProperty Size "1"}
TYPE Channel_830843C1 :
STRUCT
	{attribute addProperty Name "Input"}
	Input AT %I* : BOOL;
END_STRUCT
END_TYPE

// ---- DUTs/IO/PDOs/InfoData_6F19DB2B.TcDUT
{attribute 'GeneratedUsingTerminal: EL1809-0000-0018'}
{attribute addProperty BoxType "EL1809-0000-0018"}
{attribute addProperty Id "StateAT %I*UINT2"}
{attribute addProperty CRC "1863965483"}
{attribute addProperty Size "2"}
TYPE InfoData_6F19DB2B :
STRUCT
	{attribute addProperty Name "State"}
	State AT %I* : UINT;
END_STRUCT
END_TYPE

// ---- DUTs/IO/PDOs/Channel_42CA91F7.TcDUT
{attribute 'GeneratedUsingTerminal: EL2809-0000-0018'}
{attribute addProperty BoxType "EL2809-0000-0018"}
{attribute addProperty Id "OutputAT %Q*BOOL1"}
{attribute addProperty CRC "1120571895"}
{attribute addProperty Size "1"}
TYPE Channel_42CA91F7 :
STRUCT
	{attribute addProperty Name "Output"}
	Output AT %Q* : BOOL;
END_STRUCT
END_TYPE

// ---- DUTs/IO/PDOs/AO_Outputs_Channel_BA7EBB7C.TcDUT
{attribute 'GeneratedUsingTerminal: EL4004-0000-0020'}
{attribute addProperty BoxType "EL4004-0000-0020"}
{attribute addProperty Id "Analog_outputAT %Q*INT2"}
{attribute addProperty CRC "3128867708"}
{attribute addProperty Size "2"}
TYPE AO_Outputs_Channel_BA7EBB7C :
STRUCT
	{attribute addProperty Name "Analog_output"}
	Analog_output AT %Q* : INT;
END_STRUCT
END_TYPE

// ---- DUTs/IO/PDOs/COM_Inputs_3801C95E.TcDUT
{attribute 'GeneratedUsingTerminal: EL6001-0000-0020'}
{attribute addProperty BoxType "EL6001-0000-0020"}
{attribute addProperty Id "StatusAT %I*Status_3D84275F8Data_InAT %I*ARRAY[0..21] OF USINT22"}
{attribute addProperty CRC "1334739266"}
{attribute addProperty Size "30"}
TYPE COM_Inputs_3801C95E :
STRUCT
	{attribute addProperty Name "Status"}
	Status AT %I* : Status_3D84275F;
	{attribute addProperty Name "Data_In"}
	Data_In AT %I* : ARRAY[0..21] OF USINT;
END_STRUCT
END_TYPE

// ---- DUTs/IO/PDOs/COM_Outputs_DEF408EC.TcDUT
{attribute 'GeneratedUsingTerminal: EL6001-0000-0020'}
{attribute addProperty BoxType "EL6001-0000-0020"}
{attribute addProperty Id "CtrlAT %Q*Ctrl_71604E865Data_OutAT %Q*ARRAY[0..21] OF USINT22"}
{attribute addProperty CRC "2695605661"}
{attribute addProperty Size "27"}
TYPE COM_Outputs_DEF408EC :
STRUCT
	{attribute addProperty Name "Ctrl"}
	Ctrl AT %Q* : Ctrl_71604E86;
	{attribute addProperty Name "Data_Out"}
	Data_Out AT %Q* : ARRAY[0..21] OF USINT;
END_STRUCT
END_TYPE

// ---- DUTs/IO/PDOs/PM_Inputs_Channel_2F868086.TcDUT
{attribute 'GeneratedUsingTerminal: EL3403-0000-0023'}
{attribute addProperty BoxType "EL3403-0000-0023"}
{attribute addProperty Id "TxPDO_ToggleAT %I*BOOL1CurrentAT %I*DINT4VoltageAT %I*DINT4Active_powerAT %I*DINT4IndexAT %I*USINT1Variant_valueAT %I*DINT4"}
{attribute addProperty CRC "797343878"}
{attribute addProperty Size "18"}
TYPE PM_Inputs_Channel_2F868086 :
STRUCT
	{attribute addProperty Name "TxPDO_Toggle"}
	TxPDO_Toggle AT %I* : BOOL;
	{attribute addProperty Name "Current"}
	Current AT %I* : DINT;
	{attribute addProperty Name "Voltage"}
	Voltage AT %I* : DINT;
	{attribute addProperty Name "Active_power"}
	Active_power AT %I* : DINT;
	{attribute addProperty Name "Index"}
	Index AT %I* : USINT;
	{attribute addProperty Name "Variant_value"}
	Variant_value AT %I* : DINT;
END_STRUCT
END_TYPE

// ---- DUTs/IO/PDOs/PM_Status_data_2A9514CB.TcDUT
{attribute 'GeneratedUsingTerminal: EL3403-0000-0023'}
{attribute addProperty BoxType "EL3403-0000-0023"}
{attribute addProperty Id "Missing_zero_crossing_AAT %I*BOOL1Missing_zero_crossing_BAT %I*BOOL1Missing_zero_crossing_CAT %I*BOOL1Phase_sequence_errorAT %I*BOOL1"}
{attribute addProperty CRC "714413259"}
{attribute addProperty Size "4"}
TYPE PM_Status_data_2A9514CB :
STRUCT
	{attribute addProperty Name "Missing_zero_crossing_A"}
	Missing_zero_crossing_A AT %I* : BOOL;
	{attribute addProperty Name "Missing_zero_crossing_B"}
	Missing_zero_crossing_B AT %I* : BOOL;
	{attribute addProperty Name "Missing_zero_crossing_C"}
	Missing_zero_crossing_C AT %I* : BOOL;
	{attribute addProperty Name "Phase_sequence_error"}
	Phase_sequence_error AT %I* : BOOL;
END_STRUCT
END_TYPE

// ---- DUTs/IO/PDOs/PM_Outputs_Channel_E5FBDE30.TcDUT
{attribute 'GeneratedUsingTerminal: EL3403-0000-0023'}
{attribute addProperty BoxType "EL3403-0000-0023"}
{attribute addProperty Id "IndexAT %Q*USINT1"}
{attribute addProperty CRC "3858488880"}
{attribute addProperty Size "1"}
TYPE PM_Outputs_Channel_E5FBDE30 :
STRUCT
	{attribute addProperty Name "Index"}
	Index AT %Q* : USINT;
END_STRUCT
END_TYPE

// ---- DUTs/IO/PDOs/AI_Standard_Channel_A8DF64E3.TcDUT
{attribute 'GeneratedUsingTerminal: EL3174-0002-0017'}
{attribute addProperty BoxType "EL3174-0002-0017"}
{attribute addProperty Id "StatusAT %I*Status_B07533568ValueAT %I*INT2"}
{attribute addProperty CRC "2833212643"}
{attribute addProperty Size "10"}
TYPE AI_Standard_Channel_A8DF64E3 :
STRUCT
	{attribute addProperty Name "Status"}
	Status AT %I* : Status_B0753356;
	{attribute addProperty Name "Value"}
	Value AT %I* : INT;
END_STRUCT
END_TYPE

// ---- DUTs/IO/PDOs/AI_Standard_4A394481.TcDUT
{attribute 'GeneratedUsingTerminal: EL3011-0000-0018'}
{attribute addProperty BoxType "EL3011-0000-0018"}
{attribute addProperty Id "StatusAT %I*Status_F2CE6D917ValueAT %I*INT2"}
{attribute addProperty CRC "1245267073"}
{attribute addProperty Size "9"}
TYPE AI_Standard_4A394481 :
STRUCT
	{attribute addProperty Name "Status"}
	Status AT %I* : Status_F2CE6D91;
	{attribute addProperty Name "Value"}
	Value AT %I* : INT;
END_STRUCT
END_TYPE

// ---- DUTs/IO/PDOs/AI_Standard_Channel_4A394481.TcDUT
{attribute 'GeneratedUsingTerminal: EL3024-0000-0018'}
{attribute addProperty BoxType "EL3024-0000-0018"}
{attribute addProperty Id "StatusAT %I*Status_F2CE6D917ValueAT %I*INT2"}
{attribute addProperty CRC "1245267073"}
{attribute addProperty Size "9"}
TYPE AI_Standard_Channel_4A394481 :
STRUCT
	{attribute addProperty Name "Status"}
	Status AT %I* : Status_F2CE6D91;
	{attribute addProperty Name "Value"}
	Value AT %I* : INT;
END_STRUCT
END_TYPE

// ---- DUTs/IO/Boxes/EL6002_81703A53.TcDUT
{attribute 'GeneratedUsingTerminal: EL6002-0000-0019'}
{attribute addProperty BoxType "EL6002-0000-0019"}
{attribute addProperty Id "COM_TxPDO_Map_Inputs_Channel_1AT %I*COM_TxPDO_Map_Inputs_Channel_3801C95E30COM_TxPDO_Map_Inputs_Channel_2AT %I*COM_TxPDO_Map_Inputs_Channel_3801C95E30COM_RxPDO_Map_Outputs_Channel_1AT %Q*COM_RxPDO_Map_Outputs_Channel_EADA2E0D27COM_RxPDO_Map_Outputs_Channel_2AT %Q*COM_RxPDO_Map_Outputs_Channel_EADA2E0D27WcStateAT %I*WcState_9091E0EB2InfoDataAT %I*InfoData_32EB74EA10"}
{attribute addProperty CRC "2171615827"}
{attribute addProperty Size "126"}
TYPE EL6002_81703A53 :
STRUCT
	{attribute addProperty Name "COM_TxPDO_Map_Inputs_Channel_1"}
	COM_TxPDO_Map_Inputs_Channel_1 : COM_TxPDO_Map_Inputs_Channel_3801C95E;
	{attribute addProperty Name "COM_TxPDO_Map_Inputs_Channel_2"}
	COM_TxPDO_Map_Inputs_Channel_2 : COM_TxPDO_Map_Inputs_Channel_3801C95E;
	{attribute addProperty Name "COM_RxPDO_Map_Outputs_Channel_1"}
	COM_RxPDO_Map_Outputs_Channel_1 : COM_RxPDO_Map_Outputs_Channel_EADA2E0D;
	{attribute addProperty Name "COM_RxPDO_Map_Outputs_Channel_2"}
	COM_RxPDO_Map_Outputs_Channel_2 : COM_RxPDO_Map_Outputs_Channel_EADA2E0D;
	{attribute addProperty Name "WcState"}
	WcState : WcState_9091E0EB;
	{attribute addProperty Name "InfoData"}
	InfoData : InfoData_32EB74EA;
END_STRUCT
END_TYPE

// ---- DUTs/IO/Boxes/EL2809_2B6483BD.TcDUT
{attribute 'GeneratedUsingTerminal: EL2809-0000-0018'}
{attribute addProperty BoxType "EL2809-0000-0018"}
{attribute addProperty Id "Channel_1AT %Q*Channel_42CA91F71Channel_2AT %Q*Channel_42CA91F71Channel_3AT %Q*Channel_42CA91F71Channel_4AT %Q*Channel_42CA91F71Channel_5AT %Q*Channel_42CA91F71Channel_6AT %Q*Channel_42CA91F71Channel_7AT %Q*Channel_42CA91F71Channel_8AT %Q*Channel_42CA91F71Channel_9AT %Q*Channel_42CA91F71Channel_10AT %Q*Channel_42CA91F71Channel_11AT %Q*Channel_42CA91F71Channel_12AT %Q*Channel_42CA91F71Channel_13AT %Q*Channel_42CA91F71Channel_14AT %Q*Channel_42CA91F71Channel_15AT %Q*Channel_42CA91F71Channel_16AT %Q*Channel_42CA91F71WcStateAT %I*WcState_0B2B16F91InfoDataAT %I*InfoData_6F19DB2B2"}
{attribute addProperty CRC "728007613"}
{attribute addProperty Size "19"}
TYPE EL2809_2B6483BD :
STRUCT
	{attribute addProperty Name "Channel_1"}
	Channel_1 : Channel_42CA91F7;
	{attribute addProperty Name "Channel_2"}
	Channel_2 : Channel_42CA91F7;
	{attribute addProperty Name "Channel_3"}
	Channel_3 : Channel_42CA91F7;
	{attribute addProperty Name "Channel_4"}
	Channel_4 : Channel_42CA91F7;
	{attribute addProperty Name "Channel_5"}
	Channel_5 : Channel_42CA91F7;
	{attribute addProperty Name "Channel_6"}
	Channel_6 : Channel_42CA91F7;
	{attribute addProperty Name "Channel_7"}
	Channel_7 : Channel_42CA91F7;
	{attribute addProperty Name "Channel_8"}
	Channel_8 : Channel_42CA91F7;
	{attribute addProperty Name "Channel_9"}
	Channel_9 : Channel_42CA91F7;
	{attribute addProperty Name "Channel_10"}
	Channel_10 : Channel_42CA91F7;
	{attribute addProperty Name "Channel_11"}
	Channel_11 : Channel_42CA91F7;
	{attribute addProperty Name "Channel_12"}
	Channel_12 : Channel_42CA91F7;
	{attribute addProperty Name "Channel_13"}
	Channel_13 : Channel_42CA91F7;
	{attribute addProperty Name "Channel_14"}
	Channel_14 : Channel_42CA91F7;
	{attribute addProperty Name "Channel_15"}
	Channel_15 : Channel_42CA91F7;
	{attribute addProperty Name "Channel_16"}
	Channel_16 : Channel_42CA91F7;
	{attribute addProperty Name "WcState"}
	WcState : TcoIoBeckhoff.WcState_0B2B16F9;
	{attribute addProperty Name "InfoData"}
	InfoData : InfoData_6F19DB2B;
END_STRUCT
END_TYPE

// ---- DUTs/IO/Boxes/EL4004_D2A7C9B7.TcDUT
{attribute 'GeneratedUsingTerminal: EL4004-0000-0020'}
{attribute addProperty BoxType "EL4004-0000-0020"}
{attribute addProperty Id "AO_Outputs_Channel_1AT %Q*AO_Outputs_Channel_BA7EBB7C2AO_Outputs_Channel_2AT %Q*AO_Outputs_Channel_BA7EBB7C2AO_Outputs_Channel_3AT %Q*AO_Outputs_Channel_BA7EBB7C2AO_Outputs_Channel_4AT %Q*AO_Outputs_Channel_BA7EBB7C2WcStateAT %I*WcState_0B2B16F91InfoDataAT %I*InfoData_32EB74EA10"}
{attribute addProperty CRC "3534211511"}
{attribute addProperty Size "19"}
TYPE EL4004_D2A7C9B7 :
STRUCT
	{attribute addProperty Name "AO_Outputs_Channel_1"}
	AO_Outputs_Channel_1 : AO_Outputs_Channel_BA7EBB7C;
	{attribute addProperty Name "AO_Outputs_Channel_2"}
	AO_Outputs_Channel_2 : AO_Outputs_Channel_BA7EBB7C;
	{attribute addProperty Name "AO_Outputs_Channel_3"}
	AO_Outputs_Channel_3 : AO_Outputs_Channel_BA7EBB7C;
	{attribute addProperty Name "AO_Outputs_Channel_4"}
	AO_Outputs_Channel_4 : AO_Outputs_Channel_BA7EBB7C;
	{attribute addProperty Name "WcState"}
	WcState : TcoIoBeckhoff.WcState_0B2B16F9;
	{attribute addProperty Name "InfoData"}
	InfoData : InfoData_32EB74EA;
END_STRUCT
END_TYPE

// ---- DUTs/IO/Boxes/EL6001_B592E1CA.TcDUT
{attribute 'GeneratedUsingTerminal: EL6001-0000-0020'}
{attribute addProperty BoxType "EL6001-0000-0020"}
{attribute addProperty Id "COM_InputsAT %I*COM_Inputs_3801C95E30COM_OutputsAT %Q*COM_Outputs_DEF408EC27WcStateAT %I*WcState_9091E0EB2InfoDataAT %I*InfoData_32EB74EA10"}
{attribute addProperty CRC "3046302154"}
{attribute addProperty Size "69"}
TYPE EL6001_B592E1CA :
STRUCT
	{attribute addProperty Name "COM_Inputs"}
	COM_Inputs : COM_Inputs_3801C95E;
	{attribute addProperty Name "COM_Outputs"}
	COM_Outputs : COM_Outputs_DEF408EC;
	{attribute addProperty Name "WcState"}
	WcState : WcState_9091E0EB;
	{attribute addProperty Name "InfoData"}
	InfoData : InfoData_32EB74EA;
END_STRUCT
END_TYPE

// ---- DUTs/IO/Boxes/EL3403_200C4240.TcDUT
{attribute 'GeneratedUsingTerminal: EL3403-0000-0023'}
{attribute addProperty BoxType "EL3403-0000-0023"}
{attribute addProperty Id "PM_Inputs_Channel_1AT %I*PM_Inputs_Channel_2F86808618PM_Inputs_Channel_2AT %I*PM_Inputs_Channel_2F86808618PM_Inputs_Channel_3AT %I*PM_Inputs_Channel_2F86808618PM_Status_dataAT %I*PM_Status_data_2A9514CB4PM_Outputs_Channel_1AT %Q*PM_Outputs_Channel_E5FBDE301PM_Outputs_Channel_2AT %Q*PM_Outputs_Channel_E5FBDE301PM_Outputs_Channel_3AT %Q*PM_Outputs_Channel_E5FBDE301WcStateAT %I*WcState_9091E0EB2InfoDataAT %I*InfoData_32EB74EA10"}
{attribute addProperty CRC "537674304"}
{attribute addProperty Size "73"}
TYPE EL3403_200C4240 :
STRUCT
	{attribute addProperty Name "PM_Inputs_Channel_1"}
	PM_Inputs_Channel_1 : PM_Inputs_Channel_2F868086;
	{attribute addProperty Name "PM_Inputs_Channel_2"}
	PM_Inputs_Channel_2 : PM_Inputs_Channel_2F868086;
	{attribute addProperty Name "PM_Inputs_Channel_3"}
	PM_Inputs_Channel_3 : PM_Inputs_Channel_2F868086;
	{attribute addProperty Name "PM_Status_data"}
	PM_Status_data : PM_Status_data_2A9514CB;
	{attribute addProperty Name "PM_Outputs_Channel_1"}
	PM_Outputs_Channel_1 : PM_Outputs_Channel_E5FBDE30;
	{attribute addProperty Name "PM_Outputs_Channel_2"}
	PM_Outputs_Channel_2 : PM_Outputs_Channel_E5FBDE30;
	{attribute addProperty Name "PM_Outputs_Channel_3"}
	PM_Outputs_Channel_3 : PM_Outputs_Channel_E5FBDE30;
	{attribute addProperty Name "WcState"}
	WcState : WcState_9091E0EB;
	{attribute addProperty Name "InfoData"}
	InfoData : InfoData_32EB74EA;
END_STRUCT
END_TYPE

// ---- DUTs/IO/Boxes/EL2008_E2806B95.TcDUT
{attribute 'GeneratedUsingTerminal: EL2008-0000-0017'}
{attribute addProperty BoxType "EL2008-0000-0017"}
{attribute addProperty Id "Channel_1AT %Q*Channel_42CA91F71Channel_2AT %Q*Channel_42CA91F71Channel_3AT %Q*Channel_42CA91F71Channel_4AT %Q*Channel_42CA91F71Channel_5AT %Q*Channel_42CA91F71Channel_6AT %Q*Channel_42CA91F71Channel_7AT %Q*Channel_42CA91F71Channel_8AT %Q*Channel_42CA91F71WcStateAT %I*WcState_0B2B16F91InfoDataAT %I*InfoData_6F19DB2B2"}
{attribute addProperty CRC "3800066965"}
{attribute addProperty Size "11"}
{attribute clr [Container(Layout.Stack)]}
{attribute clr [Group(Layout.GroupBox)]}
TYPE EL2008_E2806B95 :
STRUCT
	{attribute addProperty Name "Channel_1"}
	Channel_1 : Channel_42CA91F7;
	{attribute addProperty Name "Channel_2"}
	Channel_2 : Channel_42CA91F7;
	{attribute addProperty Name "Channel_3"}
	Channel_3 : Channel_42CA91F7;
	{attribute addProperty Name "Channel_4"}
	Channel_4 : Channel_42CA91F7;
	{attribute addProperty Name "Channel_5"}
	Channel_5 : Channel_42CA91F7;
	{attribute addProperty Name "Channel_6"}
	Channel_6 : Channel_42CA91F7;
	{attribute addProperty Name "Channel_7"}
	Channel_7 : Channel_42CA91F7;
	{attribute addProperty Name "Channel_8"}
	Channel_8 : Channel_42CA91F7;
	{attribute addProperty Name "WcState"}
	WcState : TcoIoBeckhoff.WcState_0B2B16F9;
	{attribute addProperty Name "InfoData"}
	InfoData : InfoData_6F19DB2B;
END_STRUCT
END_TYPE

// ---- DUTs/IO/Devices/SyncUnitTasks_1988CF1B.TcDUT
{attribute 'GeneratedUsingTerminal: '}
{attribute addProperty BoxType ""}
{attribute addProperty Id "unreferencedAT %I*SyncUnitTask_2D604ED59PlcTaskAT %I*SyncUnitTask_2D604ED59PlcTask1AT %I*SyncUnitTask_2D604ED59PlcTask2AT %I*SyncUnitTask_2D604ED59"}
{attribute addProperty CRC "428396315"}
{attribute addProperty Size "36"}
TYPE SyncUnitTasks_1988CF1B :
STRUCT
	{attribute addProperty Name "unreferenced"}
	unreferenced : TcoIoBeckhoff.SyncUnitTask_2D604ED5;
	{attribute addProperty Name "PlcTask"}
	PlcTask : TcoIoBeckhoff.SyncUnitTask_2D604ED5;
	{attribute addProperty Name "PlcTask1"}
	PlcTask1 : TcoIoBeckhoff.SyncUnitTask_2D604ED5;
	{attribute addProperty Name "PlcTask2"}
	PlcTask2 : TcoIoBeckhoff.SyncUnitTask_2D604ED5;
END_STRUCT
END_TYPE

// ---- DUTs/IO/Devices/SyncUnits_13973095.TcDUT
{attribute 'GeneratedUsingTerminal: '}
{attribute addProperty BoxType ""}
{attribute addProperty Id "_defaultAT %I*SyncUnitTasks_1988CF1B36"}
{attribute addProperty CRC "328675477"}
{attribute addProperty Size "36"}
TYPE SyncUnits_13973095 :
STRUCT
	{attribute addProperty Name "_default"}
	_default : SyncUnitTasks_1988CF1B;
END_STRUCT
END_TYPE

// ---- DUTs/IO/Topology/Device_1_EtherCAT_4442729B.TcDUT
{attribute 'GeneratedUsingTerminal: IODEVICETYPE_ETHERCATPROT'}
{attribute addProperty BoxType "IODEVICETYPE_ETHERCATPROT"}
{attribute addProperty Id "Term_1_EK1200Term_1_EK1200_342ABB04272SyncUnitsSyncUnits_1397309536InputsInputs_A65FACA410OutputsOutputs_23C0ED1D6InfoDataInfoData_E68C61CD28"}
{attribute addProperty CRC "1145205403"}
{attribute addProperty Size "352"}
TYPE Device_1_EtherCAT_4442729B :
STRUCT
	{attribute addProperty Name "Term_1_EK1200"}
	Term_1_EK1200 : Term_1_EK1200_342ABB04;
	{attribute addProperty Name "SyncUnits"}
	SyncUnits : SyncUnits_13973095;
	{attribute addProperty Name "Inputs"}
	Inputs : TcoIoBeckhoff.Inputs_A65FACA4;
	{attribute addProperty Name "Outputs"}
	Outputs : TcoIoBeckhoff.Outputs_23C0ED1D;
	{attribute addProperty Name "InfoData"}
	InfoData : TcoIoBeckhoff.InfoData_E68C61CD;
END_STRUCT
END_TYPE

// ---- DUTs/IO/Topology/Term_9_EK1100_B6B701E6.TcDUT
{attribute 'GeneratedUsingTerminal: EK1100-0000-0018'}
{attribute addProperty BoxType "EK1100-0000-0018"}
{attribute addProperty Id "Term_10_EL6001EL6001_B592E1CA69Term_11_EL1809EL1809_32157CFD20Term_12_EL2809EL2809_2B6483BD19Term_13_EK1110EK1110_1FC0878B2"}
{attribute addProperty CRC "3065446886"}
{attribute addProperty Size "110"}
TYPE Term_9_EK1100_B6B701E6 EXTENDS TcoCore.EK1100_1FC0878B :
STRUCT
	{attribute addProperty Name "Term_10_EL6001"}
	Term_10_EL6001 : EL6001_B592E1CA;
	{attribute addProperty Name "Term_11_EL1809"}
	Term_11_EL1809 : EL1809_32157CFD;
	{attribute addProperty Name "Term_12_EL2809"}
	Term_12_EL2809 : EL2809_2B6483BD;
	{attribute addProperty Name "Term_13_EK1110"}
	Term_13_EK1110 : EK1110_1FC0878B;
END_STRUCT
END_TYPE

// ---- DUTs/IO/Topology/Device_4_EtherCAT_7DA382B8.TcDUT
{attribute 'GeneratedUsingTerminal: IODEVICETYPE_ETHERCATPROT'}
{attribute addProperty BoxType "IODEVICETYPE_ETHERCATPROT"}
{attribute addProperty Id "Term_9_EK1100Term_9_EK1100_B6B701E6110Term_14_EK1100Term_14_EK1100_ED6DF06D285SyncUnitsSyncUnits_1397309536InputsInputs_A65FACA410OutputsOutputs_23C0ED1D6InfoDataInfoData_E68C61CD28"}
{attribute addProperty CRC "2107867832"}
{attribute addProperty Size "475"}
TYPE Device_4_EtherCAT_7DA382B8 :
STRUCT
	{attribute addProperty Name "Term_9_EK1100"}
	Term_9_EK1100 : Term_9_EK1100_B6B701E6;
	{attribute addProperty Name "Term_14_EK1100"}
	Term_14_EK1100 : Term_14_EK1100_ED6DF06D;
	{attribute addProperty Name "SyncUnits"}
	SyncUnits : SyncUnits_13973095;
	{attribute addProperty Name "Inputs"}
	Inputs : TcoIoBeckhoff.Inputs_A65FACA4;
	{attribute addProperty Name "Outputs"}
	Outputs : TcoIoBeckhoff.Outputs_23C0ED1D;
	{attribute addProperty Name "InfoData"}
	InfoData : TcoIoBeckhoff.InfoData_E68C61CD;
END_STRUCT
END_TYPE

// ---- GVLs/GVL_iXlinker.TcGVL
{attribute 'qualified_only'}
VAR_GLOBAL
		Device_1_EtherCAT : Device_1_EtherCAT_B6FFA96B;
		Device_4_EtherCAT : Device_4_EtherCAT_2B006C36;
END_VAR

// ---- POUs/MAIN.TcPOU
PROGRAM MAIN
VAR
	_tcc : tcc;

END_VAR

_tcc.Run();

END_PROGRAM

// ---- POUs/tcc.TcPOU
FUNCTION_BLOCK tcc EXTENDS TcoCore.TcoContext
VAR
	{attribute addProperty Name "Device 1 (EtherCAT)"}
	Device_1 : TcoIoBeckhoff.TcoEthercatMasterDevice(THIS^);
	{attribute addProperty Name "Device 4 (EtherCAT)"}
	Device_4 : TcoIoBeckhoff.TcoEthercatMasterDevice(THIS^);
END_VAR

{attribute 'hide'}
METHOD FB_init : BOOL
VAR_INPUT
	bInitRetains : BOOL; // if TRUE, the retain variables are initialized (warm start / cold start)
	bInCopyCode : BOOL;  // if TRUE, the instance afterwards gets moved into the copy code (online change)
END_VAR
END_METHOD

(*~
	<docu>
		<summary>
			Main method of the TcoContext. This is the entry point of any control logic that belongs to this context. 
			The call of this method is ensured by calling the <c>InstanceName.Run()</c> method, and it must not be called explicitly.
			This method is abstract, and it must be overridden in derived block.
		</summary>
	</docu>
~*)
METHOD PROTECTED  Main
VAR
END_VAR
Device_1(	Inputs			:=			GVL_iXlinker.Device_1_EtherCAT.Inputs,
			InfoData		:=			GVL_iXlinker.Device_1_EtherCAT.InfoData,
			SyncUnits		:= ADR(		GVL_iXlinker.Device_1_EtherCAT.SyncUnits),
			SyncUnitsSize	:= SIZEOF(	GVL_iXlinker.Device_1_EtherCAT.SyncUnits));	

			
			
Device_4(	Inputs			:=			GVL_iXlinker.Device_4_EtherCAT.Inputs,
			InfoData		:=			GVL_iXlinker.Device_4_EtherCAT.InfoData,
			SyncUnits		:= ADR(		GVL_iXlinker.Device_4_EtherCAT.SyncUnits),
			SyncUnitsSize	:= SIZEOF(	GVL_iXlinker.Device_4_EtherCAT.SyncUnits));
END_METHOD

END_FUNCTION_BLOCK
